LIN {X 0,Y 382.992,Z 182.274,A -85,B 0,C 180,E1 -11850.301,E2 -11850.301} C_VEL
LIN {X 0,Y 383.051,Z 182.269,A -85,B 0,C 180,E1 -11852.698,E2 -11852.698} C_VEL
LIN {X 0,Y 383.046,Z 182.274,A -85,B 0,C 180,E1 -11855.04,E2 -11855.04} C_VEL
LIN {X 0,Y 382.987,Z 182.277,A -85,B 0,C 180,E1 -11858.469,E2 -11858.469} C_VEL
LIN {X 0,Y 383.057,Z 182.266,A -85,B 0,C 180,E1 -11861.827,E2 -11861.827} C_VEL
LIN {X 0,Y 383.104,Z 182.263,A -85,B 0,C 180,E1 -11865.119,E2 -11865.119} C_VEL
LIN {X 0,Y 383.092,Z 182.265,A -85,B 0,C 180,E1 -11868.358,E2 -11868.358} C_VEL
LIN {X 0,Y 383.258,Z 182.242,A -85,B 0,C 180,E1 -11871.976,E2 -11871.976} C_VEL
LIN {X 0,Y 383.192,Z 182.253,A -85,B 0,C 180,E1 -11874.739,E2 -11874.739} C_VEL
LIN {X 0,Y 383.38,Z 182.228,A -85,B 0,C 180,E1 -11877.899,E2 -11877.899} C_VEL
LIN {X 0,Y 383.514,Z 182.212,A -85,B 0,C 180,E1 -11880.001,E2 -11880.001} C_VEL
LIN {X 0,Y 383.24,Z 182.243,A -85,B 0,C 180,E1 -11883.154,E2 -11883.154} C_VEL
LIN {X 0,Y 383.275,Z 182.243,A -85,B 0,C 180,E1 -11886.317,E2 -11886.317} C_VEL
LIN {X 0,Y 383.147,Z 182.256,A -85,B 0,C 180,E1 -11889.503,E2 -11889.503} C_VEL
LIN {X 0,Y 383.121,Z 182.261,A -85,B 0,C 180,E1 -11893.537,E2 -11893.537} C_VEL
LIN {X 0,Y 383.091,Z 182.265,A -85,B 0,C 180,E1 -11897.455,E2 -11897.455} C_VEL
LIN {X 0,Y 383.025,Z 182.27,A -85,B 0,C 180,E1 -11900.648,E2 -11900.648} C_VEL
LIN {X 0,Y 383.03,Z 182.274,A -85,B 0,C 180,E1 -11903.808,E2 -11903.808} C_VEL
LIN {X 0,Y 383.077,Z 182.265,A -85,B 0,C 180,E1 -11906.124,E2 -11906.124} C_VEL
LIN {X 0,Y 382.989,Z 182.278,A -85,B 0,C 180,E1 -11909.701,E2 -11909.701} C_VEL
LIN {X 0,Y 383.001,Z 182.279,A -85,B 0,C 180,E1 -11913.402,E2 -11913.402} C_VEL
LIN {X 0,Y 383.03,Z 182.274,A -85,B 0,C 180,E1 -11916.165,E2 -11916.165} C_VEL
LIN {X 0,Y 382.999,Z 182.279,A -85,B 0,C 180,E1 -11917.905,E2 -11917.905} C_VEL
LIN {X 0,Y 383.44,Z 185.021,A -85,B 0,C 180,E1 -11921.288,E2 -11921.288} C_VEL
LIN {X 0,Y 383.849,Z 188.005,A -85,B 0,C 180,E1 -11924.435,E2 -11924.435} C_VEL
LIN {X 0,Y 384.214,Z 191.062,A -85,B 0,C 180,E1 -11927.407,E2 -11927.407} C_VEL
LIN {X 0,Y 384.098,Z 194.234,A -85,B 0,C 180,E1 -11930.219,E2 -11930.219} C_VEL
LIN {X 0,Y 383.628,Z 198.472,A -85,B 0,C 180,E1 -11933.715,E2 -11933.715} C_VEL
LIN {X 0,Y 383.22,Z 202.206,A -85,B 0,C 180,E1 -11936.621,E2 -11936.621} C_VEL
LIN {X 0,Y 382.801,Z 207.145,A -85,B 0,C 180,E1 -11940.284,E2 -11940.284} C_VEL
LIN {X 0,Y 382.559,Z 210.485,A -85,B 0,C 180,E1 -11942.66,E2 -11942.66} C_VEL
LIN {X 0,Y 382.201,Z 215.542,A -85,B 0,C 180,E1 -11946.138,E2 -11946.138} C_VEL
LIN {X 0,Y 381.971,Z 220.656,A -85,B 0,C 180,E1 -11949.538,E2 -11949.538} C_VEL
LIN {X 0,Y 381.912,Z 223.237,A -85,B 0,C 180,E1 -11951.101,E2 -11951.101} C_VEL
LIN {X 0,Y 383.988,Z 233.513,A -85,B 0,C 180,E1 -11951.545,E2 -11951.545} C_VEL
LIN {X 0,Y 385.643,Z 242.984,A -85,B 0,C 180,E1 -11952.061,E2 -11952.061} C_VEL
LIN {X 0,Y 386.917,Z 251.684,A -85,B 0,C 180,E1 -11952.631,E2 -11952.631} C_VEL
LIN {X 0,Y 387.254,Z 257.307,A -85,B 0,C 180,E1 -11953.025,E2 -11953.025} C_VEL
LIN {X 0,Y 386.212,Z 269.459,A -85,B 0,C 180,E1 -11954.024,E2 -11954.024} C_VEL
LIN {X 0,Y 385.457,Z 278.408,A -85,B 0,C 180,E1 -11954.941,E2 -11954.941} C_VEL
LIN {X 0,Y 384.668,Z 287.294,A -85,B 0,C 180,E1 -11956.04,E2 -11956.04} C_VEL
LIN {X 0,Y 384.084,Z 294.166,A -85,B 0,C 180,E1 -11957.047,E2 -11957.047} C_VEL
LIN {X 0,Y 383.433,Z 300.369,A -85,B 0,C 180,E1 -11958.1,E2 -11958.1} C_VEL
LIN {X 0,Y 382.89,Z 306.911,A -85,B 0,C 180,E1 -11959.423,E2 -11959.423} C_VEL
LIN {X 0,Y 382.464,Z 311.414,A -85,B 0,C 180,E1 -11960.481,E2 -11960.481} C_VEL
LIN {X 0,Y 382.032,Z 316.908,A -85,B 0,C 180,E1 -11962.07,E2 -11962.07} C_VEL
LIN {X 0,Y 381.793,Z 321.235,A -85,B 0,C 180,E1 -11963.659,E2 -11963.659} C_VEL
LIN {X 0,Y 381.684,Z 323.603,A -85,B 0,C 180,E1 -11964.718,E2 -11964.718} C_VEL
LIN {X 0,Y 381.643,Z 325.403,A -85,B 0,C 180,E1 -11965.776,E2 -11965.776} C_VEL
LIN {X 0,Y 381.558,Z 327.847,A -85,B 0,C 180,E1 -11967.889,E2 -11967.889} C_VEL
LIN {X 0,Y 381.591,Z 328.437,A -85,B 0,C 180,E1 -11968.945,E2 -11968.945} C_VEL
LIN {X 0,Y 381.591,Z 328.437,A -85,B 0,C 180,E1 -11971.055,E2 -11971.055} C_VEL
LIN {X 0,Y 381.558,Z 327.847,A -85,B 0,C 180,E1 -11972.111,E2 -11972.111} C_VEL
LIN {X 0,Y 381.643,Z 325.403,A -85,B 0,C 180,E1 -11974.224,E2 -11974.224} C_VEL
LIN {X 0,Y 381.694,Z 322.487,A -85,B 0,C 180,E1 -11975.797,E2 -11975.797} C_VEL
LIN {X 0,Y 381.934,Z 318.462,A -85,B 0,C 180,E1 -11977.401,E2 -11977.401} C_VEL
LIN {X 0,Y 382.305,Z 313.331,A -85,B 0,C 180,E1 -11978.99,E2 -11978.99} C_VEL
LIN {X 0,Y 382.762,Z 308.067,A -85,B 0,C 180,E1 -11980.313,E2 -11980.313} C_VEL
LIN {X 0,Y 383.283,Z 301.745,A -85,B 0,C 180,E1 -11981.636,E2 -11981.636} C_VEL
LIN {X 0,Y 383.901,Z 295.793,A -85,B 0,C 180,E1 -11982.69,E2 -11982.69} C_VEL
LIN {X 0,Y 384.517,Z 288.862,A -85,B 0,C 180,E1 -11983.745,E2 -11983.745} C_VEL
LIN {X 0,Y 385.22,Z 280.677,A -85,B 0,C 180,E1 -11984.798,E2 -11984.798} C_VEL
LIN {X 0,Y 385.952,Z 272.162,A -85,B 0,C 180,E1 -11985.716,E2 -11985.716} C_VEL
LIN {X 0,Y 386.709,Z 263.445,A -85,B 0,C 180,E1 -11986.497,E2 -11986.497} C_VEL
LIN {X 0,Y 387.26,Z 254.506,A -85,B 0,C 180,E1 -11987.164,E2 -11987.164} C_VEL
LIN {X 0,Y 385.889,Z 244.456,A -85,B 0,C 180,E1 -11987.849,E2 -11987.849} C_VEL
LIN {X 0,Y 384.09,Z 233.859,A -85,B 0,C 180,E1 -11988.437,E2 -11988.437} C_VEL
LIN {X 0,Y 381.969,Z 223.863,A -85,B 0,C 180,E1 -11988.879,E2 -11988.879} C_VEL
LIN {X 0,Y 381.882,Z 223.047,A -85,B 0,C 180,E1 -11988.926,E2 -11988.926} C_VEL
LIN {X 0,Y 382.161,Z 217.233,A -85,B 0,C 180,E1 -11992.717,E2 -11992.717} C_VEL
LIN {X 0,Y 382.421,Z 212.16,A -85,B 0,C 180,E1 -11996.171,E2 -11996.171} C_VEL
LIN {X 0,Y 382.686,Z 208.821,A -85,B 0,C 180,E1 -11998.521,E2 -11998.521} C_VEL
LIN {X 0,Y 382.931,Z 205.501,A -85,B 0,C 180,E1 -12000.923,E2 -12000.923} C_VEL
LIN {X 0,Y 383.392,Z 200.573,A -85,B 0,C 180,E1 -12004.629,E2 -12004.629} C_VEL
LIN {X 0,Y 383.871,Z 196.268,A -85,B 0,C 180,E1 -12008.07,E2 -12008.07} C_VEL
LIN {X 0,Y 384.187,Z 192.607,A -85,B 0,C 180,E1 -12011.189,E2 -12011.189} C_VEL
LIN {X 0,Y 384.182,Z 190.641,A -85,B 0,C 180,E1 -12012.967,E2 -12012.967} C_VEL
LIN {X 0,Y 383.789,Z 187.652,A -85,B 0,C 180,E1 -12015.903,E2 -12015.903} C_VEL
LIN {X 0,Y 383.412,Z 184.995,A -85,B 0,C 180,E1 -12018.723,E2 -12018.723} C_VEL
LIN {X 0,Y 383.062,Z 182.677,A -85,B 0,C 180,E1 -12021.406,E2 -12021.406} C_VEL
LIN {X 0,Y 382.992,Z 182.281,A -85,B 0,C 180,E1 -12022.73,E2 -12022.73} C_VEL
LIN {X 0,Y 383.016,Z 182.276,A -85,B 0,C 180,E1 -12025.659,E2 -12025.659} C_VEL
LIN {X 0,Y 382.98,Z 182.278,A -85,B 0,C 180,E1 -12029.081,E2 -12029.081} C_VEL
LIN {X 0,Y 383.054,Z 182.271,A -85,B 0,C 180,E1 -12032.697,E2 -12032.697} C_VEL
LIN {X 0,Y 383.049,Z 182.268,A -85,B 0,C 180,E1 -12035.039,E2 -12035.039} C_VEL
LIN {X 0,Y 382.989,Z 182.28,A -85,B 0,C 180,E1 -12038.468,E2 -12038.468} C_VEL
LIN {X 0,Y 383.059,Z 182.268,A -85,B 0,C 180,E1 -12041.826,E2 -12041.826} C_VEL
LIN {X 0,Y 383.106,Z 182.26,A -85,B 0,C 180,E1 -12045.118,E2 -12045.118} C_VEL
LIN {X 0,Y 383.093,Z 182.265,A -85,B 0,C 180,E1 -12048.357,E2 -12048.357} C_VEL
LIN {X 0,Y 383.258,Z 182.247,A -85,B 0,C 180,E1 -12051.976,E2 -12051.976} C_VEL
LIN {X 0,Y 383.191,Z 182.25,A -85,B 0,C 180,E1 -12054.738,E2 -12054.738} C_VEL
LIN {X 0,Y 383.379,Z 182.231,A -85,B 0,C 180,E1 -12057.898,E2 -12057.898} C_VEL
LIN {X 0,Y 383.514,Z 182.212,A -85,B 0,C 180,E1 -12059.999,E2 -12059.999} C_VEL
LIN {X 0,Y 383.241,Z 182.245,A -85,B 0,C 180,E1 -12063.153,E2 -12063.153} C_VEL
LIN {X 0,Y 383.255,Z 182.242,A -85,B 0,C 180,E1 -12066.635,E2 -12066.635} C_VEL
LIN {X 0,Y 383.146,Z 182.261,A -85,B 0,C 180,E1 -12069.502,E2 -12069.502} C_VEL
LIN {X 0,Y 383.119,Z 182.262,A -85,B 0,C 180,E1 -12073.536,E2 -12073.536} C_VEL
LIN {X 0,Y 383.089,Z 182.266,A -85,B 0,C 180,E1 -12077.454,E2 -12077.454} C_VEL
LIN {X 0,Y 383.022,Z 182.273,A -85,B 0,C 180,E1 -12080.647,E2 -12080.647} C_VEL
LIN {X 0,Y 383.027,Z 182.27,A -85,B 0,C 180,E1 -12083.807,E2 -12083.807} C_VEL
LIN {X 0,Y 383.074,Z 182.264,A -85,B 0,C 180,E1 -12086.123,E2 -12086.123} C_VEL
LIN {X 0,Y 383.043,Z 182.271,A -85,B 0,C 180,E1 -12088.492,E2 -12088.492} C_VEL
LIN {X 0,Y 383.005,Z 182.274,A -85,B 0,C 180,E1 -12092.149,E2 -12092.149} C_VEL
LIN {X 0,Y 383.012,Z 182.278,A -85,B 0,C 180,E1 -12094.668,E2 -12094.668} C_VEL
LIN {X 0,Y 382.997,Z 182.274,A -85,B 0,C 180,E1 -12097.904,E2 -12097.904} C_VEL
LIN {X 0,Y 383.007,Z 182.272,A -85,B 0,C 180,E1 -12101.343,E2 -12101.343} C_VEL
LIN {X 0,Y 382.991,Z 182.28,A -85,B 0,C 180,E1 -12104.303,E2 -12104.303} C_VEL
LIN {X 0,Y 383.004,Z 182.273,A -85,B 0,C 180,E1 -12107.24,E2 -12107.24} C_VEL
LIN {X 0,Y 383.011,Z 182.276,A -85,B 0,C 180,E1 -12110.413,E2 -12110.413} C_VEL
LIN {X 0,Y 383.021,Z 182.277,A -85,B 0,C 180,E1 -12114.045,E2 -12114.045} C_VEL
LIN {X 0,Y 383.032,Z 182.275,A -85,B 0,C 180,E1 -12117.853,E2 -12117.853} C_VEL
LIN {X 0,Y 383.059,Z 182.271,A -85,B 0,C 180,E1 -12121.72,E2 -12121.72} C_VEL
LIN {X 0,Y 383.048,Z 182.268,A -85,B 0,C 180,E1 -12125.04,E2 -12125.04} C_VEL
LIN {X 0,Y 382.992,Z 182.274,A -85,B 0,C 180,E1 -12128.469,E2 -12128.469} C_VEL
LIN {X 0,Y 383.085,Z 182.268,A -85,B 0,C 180,E1 -12131.828,E2 -12131.828} C_VEL
LIN {X 0,Y 383.106,Z 182.265,A -85,B 0,C 180,E1 -12135.118,E2 -12135.118} C_VEL
LIN {X 0,Y 383.094,Z 182.265,A -85,B 0,C 180,E1 -12138.358,E2 -12138.358} C_VEL
LIN {X 0,Y 383.138,Z 182.283,A -85,B 0,C 180,E1 -12139.598,E2 -12139.598} C_VEL
LIN {X 0,Y 383.814,Z 184.561,A -85,B 0,C 180,E1 -12139.95,E2 -12139.95} C_VEL
LIN {X 0,Y 385.348,Z 186.561,A -85,B 0,C 180,E1 -12140.685,E2 -12140.685} C_VEL
LIN {X 0,Y 387.436,Z 187.855,A -85,B 0,C 180,E1 -12141.656,E2 -12141.656} C_VEL
LIN {X 0,Y 388.84,Z 188.564,A -85,B 0,C 180,E1 -12142.402,E2 -12142.402} C_VEL
LIN {X 0,Y 389.96,Z 190.834,A -85,B 0,C 180,E1 -12143.142,E2 -12143.142} C_VEL
LIN {X 0,Y 391.789,Z 192.993,A -85,B 0,C 180,E1 -12144.467,E2 -12144.467} C_VEL
LIN {X 0,Y 393.422,Z 194.061,A -85,B 0,C 180,E1 -12145.902,E2 -12145.902} C_VEL
LIN {X 0,Y 394.945,Z 194.431,A -85,B 0,C 180,E1 -12147.96,E2 -12147.96} C_VEL
LIN {X 0,Y 395.509,Z 194.494,A -85,B 0,C 180,E1 -12150,E2 -12150} C_VEL
LIN {X 0,Y 394.945,Z 194.431,A -85,B 0,C 180,E1 -12152.04,E2 -12152.04} C_VEL
LIN {X 0,Y 393.422,Z 194.061,A -85,B 0,C 180,E1 -12154.098,E2 -12154.098} C_VEL
LIN {X 0,Y 391.446,Z 192.7,A -85,B 0,C 180,E1 -12155.796,E2 -12155.796} C_VEL
LIN {X 0,Y 389.552,Z 190.154,A -85,B 0,C 180,E1 -12157.135,E2 -12157.135} C_VEL
LIN {X 0,Y 388.788,Z 188.398,A -85,B 0,C 180,E1 -12157.634,E2 -12157.634} C_VEL
LIN {X 0,Y 385.958,Z 187.055,A -85,B 0,C 180,E1 -12159.036,E2 -12159.036} C_VEL
LIN {X 0,Y 384.054,Z 184.967,A -85,B 0,C 180,E1 -12159.938,E2 -12159.938} C_VEL
LIN {X 0,Y 383.253,Z 182.924,A -85,B 0,C 180,E1 -12160.332,E2 -12160.332} C_VEL
LIN {X 0,Y 383.121,Z 182.263,A -85,B 0,C 180,E1 -12160.436,E2 -12160.436} C_VEL
LIN {X 0,Y 383.123,Z 182.262,A -85,B 0,C 180,E1 -12163.796,E2 -12163.796} C_VEL
LIN {X 0,Y 383.091,Z 182.267,A -85,B 0,C 180,E1 -12167.455,E2 -12167.455} C_VEL
LIN {X 0,Y 383.03,Z 182.273,A -85,B 0,C 180,E1 -12170.649,E2 -12170.649} C_VEL
LIN {X 0,Y 383.029,Z 182.271,A -85,B 0,C 180,E1 -12173.807,E2 -12173.807} C_VEL
LIN {X 0,Y 383.052,Z 182.267,A -85,B 0,C 180,E1 -12177.302,E2 -12177.302} C_VEL
LIN {X 0,Y 382.991,Z 182.275,A -85,B 0,C 180,E1 -12180.917,E2 -12180.917} C_VEL
LIN {X 0,Y 383.013,Z 182.274,A -85,B 0,C 180,E1 -12184.34,E2 -12184.34} C_VEL
LIN {X 0,Y 382.994,Z 182.275,A -85,B 0,C 180,E1 -12185.374,E2 -12185.374} C_VEL
LIN {X 0,Y 382.353,Z 182.361,A -85,B 0,C 180,E1 -12186.252,E2 -12186.252} C_VEL
LIN {X 0,Y 379.545,Z 182.717,A -85,B 0,C 180,E1 -12187.68,E2 -12187.68} C_VEL
LIN {X 0,Y 377.141,Z 183.016,A -85,B 0,C 180,E1 -12188.835,E2 -12188.835} C_VEL
LIN {X 0,Y 376.086,Z 183.142,A -85,B 0,C 180,E1 -12189.727,E2 -12189.727} C_VEL
LIN {X 0,Y 375.988,Z 183.151,A -85,B 0,C 180,E1 -12190.029,E2 -12190.029} C_VEL
LIN {X 0,Y 375.934,Z 183.159,A -85,B 0,C 180,E1 -12193.765,E2 -12193.765} C_VEL
LIN {X 0,Y 375.955,Z 183.156,A -85,B 0,C 180,E1 -12197.704,E2 -12197.704} C_VEL
LIN {X 0,Y 375.963,Z 183.15,A -85,B 0,C 180,E1 -12200.538,E2 -12200.538} C_VEL
LIN {X 0,Y 375.959,Z 183.156,A -85,B 0,C 180,E1 -12203.495,E2 -12203.495} C_VEL
LIN {X 0,Y 375.954,Z 183.152,A -85,B 0,C 180,E1 -12205.889,E2 -12205.889} C_VEL
LIN {X 0,Y 375.962,Z 183.152,A -85,B 0,C 180,E1 -12209.688,E2 -12209.688} C_VEL
LIN {X 0,Y 375.996,Z 183.146,A -85,B 0,C 180,E1 -12212.142,E2 -12212.142} C_VEL
LIN {X 0,Y 376,Z 183.147,A -85,B 0,C 180,E1 -12214.539,E2 -12214.539} C_VEL
LIN {X 0,Y 375.957,Z 183.151,A -85,B 0,C 180,E1 -12218.046,E2 -12218.046} C_VEL
LIN {X 0,Y 376.003,Z 183.146,A -85,B 0,C 180,E1 -12221.474,E2 -12221.474} C_VEL
LIN {X 0,Y 376.052,Z 183.145,A -85,B 0,C 180,E1 -12224.833,E2 -12224.833} C_VEL
LIN {X 0,Y 376.044,Z 183.141,A -85,B 0,C 180,E1 -12228.137,E2 -12228.137} C_VEL
LIN {X 0,Y 376.214,Z 183.119,A -85,B 0,C 180,E1 -12231.919,E2 -12231.919} C_VEL
LIN {X 0,Y 376.165,Z 183.129,A -85,B 0,C 180,E1 -12234.64,E2 -12234.64} C_VEL
LIN {X 0,Y 376.346,Z 183.104,A -85,B 0,C 180,E1 -12237.86,E2 -12237.86} C_VEL
LIN {X 0,Y 376.483,Z 183.088,A -85,B 0,C 180,E1 -12240.001,E2 -12240.001} C_VEL
LIN {X 0,Y 376.179,Z 183.123,A -85,B 0,C 180,E1 -12243.214,E2 -12243.214} C_VEL
LIN {X 0,Y 376.233,Z 183.119,A -85,B 0,C 180,E1 -12246.436,E2 -12246.436} C_VEL
LIN {X 0,Y 376.114,Z 183.134,A -85,B 0,C 180,E1 -12249.682,E2 -12249.682} C_VEL
LIN {X 0,Y 376.085,Z 183.138,A -85,B 0,C 180,E1 -12253.658,E2 -12253.658} C_VEL
LIN {X 0,Y 376.039,Z 183.145,A -85,B 0,C 180,E1 -12257.608,E2 -12257.608} C_VEL
LIN {X 0,Y 375.975,Z 183.149,A -85,B 0,C 180,E1 -12260.833,E2 -12260.833} C_VEL
LIN {X 0,Y 375.991,Z 183.147,A -85,B 0,C 180,E1 -12264.282,E2 -12264.282} C_VEL
LIN {X 0,Y 376.017,Z 183.143,A -85,B 0,C 180,E1 -12266.653,E2 -12266.653} C_VEL
LIN {X 0,Y 375.962,Z 183.15,A -85,B 0,C 180,E1 -12270.313,E2 -12270.313} C_VEL
LIN {X 0,Y 375.958,Z 183.155,A -85,B 0,C 180,E1 -12274.112,E2 -12274.112} C_VEL
LIN {X 0,Y 375.951,Z 183.158,A -85,B 0,C 180,E1 -12276.742,E2 -12276.742} C_VEL
LIN {X 0,Y 376.023,Z 183.591,A -85,B 0,C 180,E1 -12278.281,E2 -12278.281} C_VEL
LIN {X 0,Y 376.47,Z 186.515,A -85,B 0,C 180,E1 -12281.693,E2 -12281.693} C_VEL
LIN {X 0,Y 376.906,Z 189.765,A -85,B 0,C 180,E1 -12285.119,E2 -12285.119} C_VEL
LIN {X 0,Y 377.168,Z 192.589,A -85,B 0,C 180,E1 -12287.871,E2 -12287.871} C_VEL
LIN {X 0,Y 376.988,Z 195.718,A -85,B 0,C 180,E1 -12290.666,E2 -12290.666} C_VEL
LIN {X 0,Y 376.631,Z 198.928,A -85,B 0,C 180,E1 -12293.359,E2 -12293.359} C_VEL
LIN {X 0,Y 376.25,Z 202.125,A -85,B 0,C 180,E1 -12295.919,E2 -12295.919} C_VEL
LIN {X 0,Y 375.826,Z 207.042,A -85,B 0,C 180,E1 -12299.676,E2 -12299.676} C_VEL
LIN {X 0,Y 375.556,Z 210.367,A -85,B 0,C 180,E1 -12302.106,E2 -12302.106} C_VEL
LIN {X 0,Y 375.158,Z 215.391,A -85,B 0,C 180,E1 -12305.661,E2 -12305.661} C_VEL
LIN {X 0,Y 375.007,Z 218.771,A -85,B 0,C 180,E1 -12307.987,E2 -12307.987} C_VEL
LIN {X 0,Y 374.836,Z 222.855,A -85,B 0,C 180,E1 -12310.722,E2 -12310.722} C_VEL
LIN {X 0,Y 377.036,Z 233.737,A -85,B 0,C 180,E1 -12311.209,E2 -12311.209} C_VEL
LIN {X 0,Y 378.619,Z 242.764,A -85,B 0,C 180,E1 -12311.717,E2 -12311.717} C_VEL
LIN {X 0,Y 379.924,Z 251.828,A -85,B 0,C 180,E1 -12312.326,E2 -12312.326} C_VEL
LIN {X 0,Y 380.448,Z 257.164,A -85,B 0,C 180,E1 -12312.717,E2 -12312.717} C_VEL
LIN {X 0,Y 379.377,Z 269.247,A -85,B 0,C 180,E1 -12313.729,E2 -12313.729} C_VEL
LIN {X 0,Y 378.587,Z 278.196,A -85,B 0,C 180,E1 -12314.661,E2 -12314.661} C_VEL
LIN {X 0,Y 377.873,Z 285.861,A -85,B 0,C 180,E1 -12315.609,E2 -12315.609} C_VEL
LIN {X 0,Y 377.152,Z 293.954,A -85,B 0,C 180,E1 -12316.805,E2 -12316.805} C_VEL
LIN {X 0,Y 376.469,Z 300.157,A -85,B 0,C 180,E1 -12317.877,E2 -12317.877} C_VEL
LIN {X 0,Y 375.853,Z 306.698,A -85,B 0,C 180,E1 -12319.223,E2 -12319.223} C_VEL
LIN {X 0,Y 375.451,Z 311.202,A -85,B 0,C 180,E1 -12320.301,E2 -12320.301} C_VEL
LIN {X 0,Y 374.964,Z 316.695,A -85,B 0,C 180,E1 -12321.919,E2 -12321.919} C_VEL
LIN {X 0,Y 374.72,Z 321.023,A -85,B 0,C 180,E1 -12323.539,E2 -12323.539} C_VEL
LIN {X 0,Y 374.591,Z 323.391,A -85,B 0,C 180,E1 -12324.617,E2 -12324.617} C_VEL
LIN {X 0,Y 374.57,Z 325.192,A -85,B 0,C 180,E1 -12325.696,E2 -12325.696} C_VEL
LIN {X 0,Y 374.458,Z 327.636,A -85,B 0,C 180,E1 -12327.849,E2 -12327.849} C_VEL
LIN {X 0,Y 374.492,Z 328.226,A -85,B 0,C 180,E1 -12328.925,E2 -12328.925} C_VEL
LIN {X 0,Y 374.492,Z 328.226,A -85,B 0,C 180,E1 -12331.075,E2 -12331.075} C_VEL
LIN {X 0,Y 374.458,Z 327.636,A -85,B 0,C 180,E1 -12332.151,E2 -12332.151} C_VEL
LIN {X 0,Y 374.571,Z 325.192,A -85,B 0,C 180,E1 -12334.304,E2 -12334.304} C_VEL
LIN {X 0,Y 374.592,Z 323.391,A -85,B 0,C 180,E1 -12335.383,E2 -12335.383} C_VEL
LIN {X 0,Y 374.77,Z 319.781,A -85,B 0,C 180,E1 -12337.001,E2 -12337.001} C_VEL
LIN {X 0,Y 375.102,Z 315.034,A -85,B 0,C 180,E1 -12338.62,E2 -12338.62} C_VEL
LIN {X 0,Y 375.631,Z 309.01,A -85,B 0,C 180,E1 -12340.238,E2 -12340.238} C_VEL
LIN {X 0,Y 376.18,Z 302.91,A -85,B 0,C 180,E1 -12341.586,E2 -12341.586} C_VEL
LIN {X 0,Y 376.78,Z 297.208,A -85,B 0,C 180,E1 -12342.66,E2 -12342.66} C_VEL
LIN {X 0,Y 377.594,Z 288.65,A -85,B 0,C 180,E1 -12344.002,E2 -12344.002} C_VEL
LIN {X 0,Y 378.322,Z 280.465,A -85,B 0,C 180,E1 -12345.074,E2 -12345.074} C_VEL
LIN {X 0,Y 379.122,Z 271.951,A -85,B 0,C 180,E1 -12346.006,E2 -12346.006} C_VEL
LIN {X 0,Y 379.889,Z 263.233,A -85,B 0,C 180,E1 -12346.802,E2 -12346.802} C_VEL
LIN {X 0,Y 380.447,Z 255.846,A -85,B 0,C 180,E1 -12347.374,E2 -12347.374} C_VEL
LIN {X 0,Y 378.927,Z 244.579,A -85,B 0,C 180,E1 -12348.17,E2 -12348.17} C_VEL
LIN {X 0,Y 377.133,Z 234.279,A -85,B 0,C 180,E1 -12348.764,E2 -12348.764} C_VEL
LIN {X 0,Y 374.92,Z 223.683,A -85,B 0,C 180,E1 -12349.247,E2 -12349.247} C_VEL
LIN {X 0,Y 374.843,Z 222.829,A -85,B 0,C 180,E1 -12349.296,E2 -12349.296} C_VEL
LIN {X 0,Y 375.117,Z 216.798,A -85,B 0,C 180,E1 -12353.358,E2 -12353.358} C_VEL
LIN {X 0,Y 375.389,Z 212.026,A -85,B 0,C 180,E1 -12356.7,E2 -12356.7} C_VEL
LIN {X 0,Y 375.823,Z 207.042,A -85,B 0,C 180,E1 -12360.325,E2 -12360.325} C_VEL
LIN {X 0,Y 376.249,Z 202.125,A -85,B 0,C 180,E1 -12364.081,E2 -12364.081} C_VEL
LIN {X 0,Y 376.634,Z 198.901,A -85,B 0,C 180,E1 -12366.663,E2 -12366.663} C_VEL
LIN {X 0,Y 377.086,Z 194.756,A -85,B 0,C 180,E1 -12370.168,E2 -12370.168} C_VEL
LIN {X 0,Y 377.164,Z 192.57,A -85,B 0,C 180,E1 -12372.129,E2 -12372.129} C_VEL
LIN {X 0,Y 376.867,Z 189.497,A -85,B 0,C 180,E1 -12375.124,E2 -12375.124} C_VEL
LIN {X 0,Y 376.447,Z 186.513,A -85,B 0,C 180,E1 -12378.31,E2 -12378.31} C_VEL
LIN {X 0,Y 376.023,Z 183.598,A -85,B 0,C 180,E1 -12381.719,E2 -12381.719} C_VEL
LIN {X 0,Y 375.961,Z 183.151,A -85,B 0,C 180,E1 -12383.495,E2 -12383.495} C_VEL
LIN {X 0,Y 375.958,Z 183.154,A -85,B 0,C 180,E1 -12385.888,E2 -12385.888} C_VEL
LIN {X 0,Y 375.962,Z 183.15,A -85,B 0,C 180,E1 -12389.687,E2 -12389.687} C_VEL
LIN {X 0,Y 376.017,Z 183.143,A -85,B 0,C 180,E1 -12393.347,E2 -12393.347} C_VEL
LIN {X 0,Y 375.993,Z 183.148,A -85,B 0,C 180,E1 -12396.888,E2 -12396.888} C_VEL
LIN {X 0,Y 375.995,Z 183.152,A -85,B 0,C 180,E1 -12400.339,E2 -12400.339} C_VEL
LIN {X 0,Y 376.025,Z 183.144,A -85,B 0,C 180,E1 -12403.718,E2 -12403.718} C_VEL
LIN {X 0,Y 376.099,Z 183.133,A -85,B 0,C 180,E1 -12407.041,E2 -12407.041} C_VEL
LIN {X 0,Y 376.114,Z 183.134,A -85,B 0,C 180,E1 -12410.318,E2 -12410.318} C_VEL
LIN {X 0,Y 376.233,Z 183.119,A -85,B 0,C 180,E1 -12413.564,E2 -12413.564} C_VEL
LIN {X 0,Y 376.345,Z 183.108,A -85,B 0,C 180,E1 -12417.859,E2 -12417.859} C_VEL
LIN {X 0,Y 376.483,Z 183.088,A -85,B 0,C 180,E1 -12419.999,E2 -12419.999} C_VEL
LIN {X 0,Y 376.18,Z 183.125,A -85,B 0,C 180,E1 -12423.212,E2 -12423.212} C_VEL
LIN {X 0,Y 376.22,Z 183.118,A -85,B 0,C 180,E1 -12426.624,E2 -12426.624} C_VEL
LIN {X 0,Y 376.113,Z 183.135,A -85,B 0,C 180,E1 -12429.681,E2 -12429.681} C_VEL
LIN {X 0,Y 376.084,Z 183.137,A -85,B 0,C 180,E1 -12433.657,E2 -12433.657} C_VEL
LIN {X 0,Y 376.037,Z 183.143,A -85,B 0,C 180,E1 -12437.606,E2 -12437.606} C_VEL
LIN {X 0,Y 375.972,Z 183.153,A -85,B 0,C 180,E1 -12440.832,E2 -12440.832} C_VEL
LIN {X 0,Y 375.988,Z 183.147,A -85,B 0,C 180,E1 -12444.281,E2 -12444.281} C_VEL
LIN {X 0,Y 376.014,Z 183.147,A -85,B 0,C 180,E1 -12446.652,E2 -12446.652} C_VEL
LIN {X 0,Y 375.97,Z 183.153,A -85,B 0,C 180,E1 -12449.078,E2 -12449.078} C_VEL
LIN {X 0,Y 375.943,Z 183.158,A -85,B 0,C 180,E1 -12452.828,E2 -12452.828} C_VEL
LIN {X 0,Y 375.952,Z 183.152,A -85,B 0,C 180,E1 -12455.415,E2 -12455.415} C_VEL
LIN {X 0,Y 375.972,Z 183.152,A -85,B 0,C 180,E1 -12458.271,E2 -12458.271} C_VEL
LIN {X 0,Y 375.954,Z 183.151,A -85,B 0,C 180,E1 -12461.605,E2 -12461.605} C_VEL
LIN {X 0,Y 375.921,Z 183.155,A -85,B 0,C 180,E1 -12465.269,E2 -12465.269} C_VEL
LIN {X 0,Y 375.929,Z 183.159,A -85,B 0,C 180,E1 -12468.399,E2 -12468.399} C_VEL
LIN {X 0,Y 375.971,Z 183.151,A -85,B 0,C 180,E1 -12471.729,E2 -12471.729} C_VEL
LIN {X 0,Y 375.975,Z 183.149,A -85,B 0,C 180,E1 -12475.333,E2 -12475.333} C_VEL
LIN {X 0,Y 375.971,Z 183.151,A -85,B 0,C 180,E1 -12478.44,E2 -12478.44} C_VEL
LIN {X 0,Y 375.998,Z 183.149,A -85,B 0,C 180,E1 -12482.142,E2 -12482.142} C_VEL
LIN {X 0,Y 376.002,Z 183.145,A -85,B 0,C 180,E1 -12484.539,E2 -12484.539} C_VEL
LIN {X 0,Y 375.961,Z 183.153,A -85,B 0,C 180,E1 -12488.046,E2 -12488.046} C_VEL
LIN {X 0,Y 376.02,Z 183.148,A -85,B 0,C 180,E1 -12491.474,E2 -12491.474} C_VEL
LIN {X 0,Y 376.055,Z 183.144,A -85,B 0,C 180,E1 -12494.833,E2 -12494.833} C_VEL
LIN {X 0,Y 376.117,Z 183.315,A -85,B 0,C 180,E1 -12497.317,E2 -12497.317} C_VEL
LIN {X 0,Y 376.774,Z 185.472,A -85,B 0,C 180,E1 -12497.613,E2 -12497.613} C_VEL
LIN {X 0,Y 378.391,Z 187.585,A -85,B 0,C 180,E1 -12498.211,E2 -12498.211} C_VEL
LIN {X 0,Y 380.855,Z 188.996,A -85,B 0,C 180,E1 -12499.097,E2 -12499.097} C_VEL
LIN {X 0,Y 381.348,Z 189.793,A -85,B 0,C 180,E1 -12499.313,E2 -12499.313} C_VEL
LIN {X 0,Y 382.988,Z 192.386,A -85,B 0,C 180,E1 -12500.027,E2 -12500.027} C_VEL
LIN {X 0,Y 385.299,Z 194.35,A -85,B 0,C 180,E1 -12501.081,E2 -12501.081} C_VEL
LIN {X 0,Y 387.405,Z 195.44,A -85,B 0,C 180,E1 -12502.125,E2 -12502.125} C_VEL
LIN {X 0,Y 388.935,Z 197.999,A -85,B 0,C 180,E1 -12503.079,E2 -12503.079} C_VEL
LIN {X 0,Y 390.889,Z 200.077,A -85,B 0,C 180,E1 -12504.454,E2 -12504.454} C_VEL
LIN {X 0,Y 392.534,Z 201.093,A -85,B 0,C 180,E1 -12505.893,E2 -12505.893} C_VEL
LIN {X 0,Y 394.082,Z 201.477,A -85,B 0,C 180,E1 -12507.956,E2 -12507.956} C_VEL
LIN {X 0,Y 394.645,Z 201.533,A -85,B 0,C 180,E1 -12510,E2 -12510} C_VEL
LIN {X 0,Y 394.082,Z 201.477,A -85,B 0,C 180,E1 -12512.044,E2 -12512.044} C_VEL
LIN {X 0,Y 392.534,Z 201.093,A -85,B 0,C 180,E1 -12514.107,E2 -12514.107} C_VEL
LIN {X 0,Y 390.529,Z 199.798,A -85,B 0,C 180,E1 -12515.81,E2 -12515.81} C_VEL
LIN {X 0,Y 388.397,Z 197.203,A -85,B 0,C 180,E1 -12517.277,E2 -12517.277} C_VEL
LIN {X 0,Y 387.178,Z 195.131,A -85,B 0,C 180,E1 -12518.008,E2 -12518.008} C_VEL
LIN {X 0,Y 384.673,Z 193.95,A -85,B 0,C 180,E1 -12519.199,E2 -12519.199} C_VEL
LIN {X 0,Y 382.482,Z 191.776,A -85,B 0,C 180,E1 -12520.187,E2 -12520.187} C_VEL
LIN {X 0,Y 381.134,Z 189.202,A -85,B 0,C 180,E1 -12520.792,E2 -12520.792} C_VEL
LIN {X 0,Y 378.391,Z 187.585,A -85,B 0,C 180,E1 -12521.789,E2 -12521.789} C_VEL
LIN {X 0,Y 376.728,Z 185.375,A -85,B 0,C 180,E1 -12522.405,E2 -12522.405} C_VEL
LIN {X 0,Y 376.108,Z 183.138,A -85,B 0,C 180,E1 -12522.717,E2 -12522.717} C_VEL
LIN {X 0,Y 376.025,Z 183.147,A -85,B 0,C 180,E1 -12526.281,E2 -12526.281} C_VEL
LIN {X 0,Y 375.996,Z 183.148,A -85,B 0,C 180,E1 -12529.66,E2 -12529.66} C_VEL
LIN {X 0,Y 375.991,Z 183.147,A -85,B 0,C 180,E1 -12533.667,E2 -12533.667} C_VEL
LIN {X 0,Y 376.015,Z 183.145,A -85,B 0,C 180,E1 -12536.652,E2 -12536.652} C_VEL
LIN {X 0,Y 375.972,Z 183.149,A -85,B 0,C 180,E1 -12539.078,E2 -12539.078} C_VEL
LIN {X 0,Y 375.953,Z 183.151,A -85,B 0,C 180,E1 -12542.828,E2 -12542.828} C_VEL
LIN {X 0,Y 375.953,Z 183.153,A -85,B 0,C 180,E1 -12545.415,E2 -12545.415} C_VEL
LIN {X 0,Y 375.972,Z 183.151,A -85,B 0,C 180,E1 -12548.271,E2 -12548.271} C_VEL
LIN {X 0,Y 375.988,Z 183.151,A -85,B 0,C 180,E1 -12550.029,E2 -12550.029} C_VEL
LIN {X 0,Y 375.276,Z 183.236,A -85,B 0,C 180,E1 -12550.922,E2 -12550.922} C_VEL
LIN {X 0,Y 372.37,Z 183.598,A -85,B 0,C 180,E1 -12552.375,E2 -12552.375} C_VEL
LIN {X 0,Y 369.949,Z 183.904,A -85,B 0,C 180,E1 -12553.549,E2 -12553.549} C_VEL
LIN {X 0,Y 368.939,Z 184.025,A -85,B 0,C 180,E1 -12554.458,E2 -12554.458} C_VEL
LIN {X 0,Y 368.871,Z 184.033,A -85,B 0,C 180,E1 -12554.765,E2 -12554.765} C_VEL
LIN {X 0,Y 368.904,Z 184.03,A -85,B 0,C 180,E1 -12558.181,E2 -12558.181} C_VEL
LIN {X 0,Y 368.908,Z 184.034,A -85,B 0,C 180,E1 -12561.359,E2 -12561.359} C_VEL
LIN {X 0,Y 368.931,Z 184.03,A -85,B 0,C 180,E1 -12565.147,E2 -12565.147} C_VEL
LIN {X 0,Y 368.923,Z 184.031,A -85,B 0,C 180,E1 -12569.047,E2 -12569.047} C_VEL
LIN {X 0,Y 368.981,Z 184.022,A -85,B 0,C 180,E1 -12571.565,E2 -12571.565} C_VEL
LIN {X 0,Y 368.951,Z 184.028,A -85,B 0,C 180,E1 -12575.225,E2 -12575.225} C_VEL
LIN {X 0,Y 368.932,Z 184.032,A -85,B 0,C 180,E1 -12578.974,E2 -12578.974} C_VEL
LIN {X 0,Y 368.985,Z 184.02,A -85,B 0,C 180,E1 -12582.258,E2 -12582.258} C_VEL
LIN {X 0,Y 369.031,Z 184.015,A -85,B 0,C 180,E1 -12586.228,E2 -12586.228} C_VEL
LIN {X 0,Y 369.062,Z 184.011,A -85,B 0,C 180,E1 -12590.132,E2 -12590.132} C_VEL
LIN {X 0,Y 369.195,Z 183.993,A -85,B 0,C 180,E1 -12593.442,E2 -12593.442} C_VEL
LIN {X 0,Y 369.311,Z 183.98,A -85,B 0,C 180,E1 -12597.819,E2 -12597.819} C_VEL
LIN {X 0,Y 369.453,Z 183.964,A -85,B 0,C 180,E1 -12600.001,E2 -12600.001} C_VEL
LIN {X 0,Y 369.311,Z 183.984,A -85,B 0,C 180,E1 -12602.182,E2 -12602.182} C_VEL
LIN {X 0,Y 369.194,Z 183.995,A -85,B 0,C 180,E1 -12606.559,E2 -12606.559} C_VEL
LIN {X 0,Y 369.063,Z 184.014,A -85,B 0,C 180,E1 -12609.869,E2 -12609.869} C_VEL
LIN {X 0,Y 369.033,Z 184.018,A -85,B 0,C 180,E1 -12613.773,E2 -12613.773} C_VEL
LIN {X 0,Y 368.998,Z 184.024,A -85,B 0,C 180,E1 -12617.769,E2 -12617.769} C_VEL
LIN {X 0,Y 368.926,Z 184.028,A -85,B 0,C 180,E1 -12621.22,E2 -12621.22} C_VEL
LIN {X 0,Y 368.955,Z 184.023,A -85,B 0,C 180,E1 -12624.776,E2 -12624.776} C_VEL
LIN {X 0,Y 368.96,Z 184.025,A -85,B 0,C 180,E1 -12627.204,E2 -12627.204} C_VEL
LIN {X 0,Y 368.927,Z 184.028,A -85,B 0,C 180,E1 -12630.954,E2 -12630.954} C_VEL
LIN {X 0,Y 368.927,Z 184.032,A -85,B 0,C 180,E1 -12635.002,E2 -12635.002} C_VEL
LIN {X 0,Y 368.932,Z 184.199,A -85,B 0,C 180,E1 -12637.56,E2 -12637.56} C_VEL
LIN {X 0,Y 369.295,Z 186.54,A -85,B 0,C 180,E1 -12640.428,E2 -12640.428} C_VEL
LIN {X 0,Y 369.713,Z 189.523,A -85,B 0,C 180,E1 -12643.752,E2 -12643.752} C_VEL
LIN {X 0,Y 370.091,Z 192.578,A -85,B 0,C 180,E1 -12646.872,E2 -12646.872} C_VEL
LIN {X 0,Y 370.058,Z 195.691,A -85,B 0,C 180,E1 -12649.781,E2 -12649.781} C_VEL
LIN {X 0,Y 369.614,Z 199.396,A -85,B 0,C 180,E1 -12652.998,E2 -12652.998} C_VEL
LIN {X 0,Y 369.105,Z 203.672,A -85,B 0,C 180,E1 -12656.484,E2 -12656.484} C_VEL
LIN {X 0,Y 368.666,Z 208.579,A -85,B 0,C 180,E1 -12660.288,E2 -12660.288} C_VEL
LIN {X 0,Y 368.3,Z 213.278,A -85,B 0,C 180,E1 -12663.75,E2 -12663.75} C_VEL
LIN {X 0,Y 367.948,Z 218.597,A -85,B 0,C 180,E1 -12667.542,E2 -12667.542} C_VEL
LIN {X 0,Y 367.76,Z 222.609,A -85,B 0,C 180,E1 -12670.318,E2 -12670.318} C_VEL
LIN {X 0,Y 370.839,Z 237.835,A -85,B 0,C 180,E1 -12671.063,E2 -12671.063} C_VEL
LIN {X 0,Y 372.833,Z 250.677,A -85,B 0,C 180,E1 -12671.913,E2 -12671.913} C_VEL
LIN {X 0,Y 373.587,Z 258.125,A -85,B 0,C 180,E1 -12672.483,E2 -12672.483} C_VEL
LIN {X 0,Y 372.554,Z 269.036,A -85,B 0,C 180,E1 -12673.422,E2 -12673.422} C_VEL
LIN {X 0,Y 371.714,Z 277.984,A -85,B 0,C 180,E1 -12674.37,E2 -12674.37} C_VEL
LIN {X 0,Y 370.942,Z 286.001,A -85,B 0,C 180,E1 -12675.386,E2 -12675.386} C_VEL
LIN {X 0,Y 370.226,Z 293.743,A -85,B 0,C 180,E1 -12676.553,E2 -12676.553} C_VEL
LIN {X 0,Y 369.518,Z 299.945,A -85,B 0,C 180,E1 -12677.645,E2 -12677.645} C_VEL
LIN {X 0,Y 368.831,Z 306.485,A -85,B 0,C 180,E1 -12679.015,E2 -12679.015} C_VEL
LIN {X 0,Y 368.414,Z 310.99,A -85,B 0,C 180,E1 -12680.114,E2 -12680.114} C_VEL
LIN {X 0,Y 367.911,Z 316.483,A -85,B 0,C 180,E1 -12681.763,E2 -12681.763} C_VEL
LIN {X 0,Y 367.644,Z 320.811,A -85,B 0,C 180,E1 -12683.414,E2 -12683.414} C_VEL
LIN {X 0,Y 367.507,Z 323.179,A -85,B 0,C 180,E1 -12684.513,E2 -12684.513} C_VEL
LIN {X 0,Y 367.476,Z 324.98,A -85,B 0,C 180,E1 -12685.613,E2 -12685.613} C_VEL
LIN {X 0,Y 367.359,Z 327.424,A -85,B 0,C 180,E1 -12687.807,E2 -12687.807} C_VEL
LIN {X 0,Y 367.392,Z 328.015,A -85,B 0,C 180,E1 -12688.904,E2 -12688.904} C_VEL
LIN {X 0,Y 367.392,Z 328.015,A -85,B 0,C 180,E1 -12691.096,E2 -12691.096} C_VEL
LIN {X 0,Y 367.359,Z 327.424,A -85,B 0,C 180,E1 -12692.193,E2 -12692.193} C_VEL
LIN {X 0,Y 367.477,Z 324.98,A -85,B 0,C 180,E1 -12694.387,E2 -12694.387} C_VEL
LIN {X 0,Y 367.552,Z 321.85,A -85,B 0,C 180,E1 -12696.117,E2 -12696.117} C_VEL
LIN {X 0,Y 367.793,Z 318.038,A -85,B 0,C 180,E1 -12697.687,E2 -12697.687} C_VEL
LIN {X 0,Y 368.231,Z 312.906,A -85,B 0,C 180,E1 -12699.336,E2 -12699.336} C_VEL
LIN {X 0,Y 368.75,Z 307.643,A -85,B 0,C 180,E1 -12700.709,E2 -12700.709} C_VEL
LIN {X 0,Y 369.337,Z 301.321,A -85,B 0,C 180,E1 -12702.082,E2 -12702.082} C_VEL
LIN {X 0,Y 370.031,Z 295.37,A -85,B 0,C 180,E1 -12703.174,E2 -12703.174} C_VEL
LIN {X 0,Y 370.844,Z 287.174,A -85,B 0,C 180,E1 -12704.447,E2 -12704.447} C_VEL
LIN {X 0,Y 371.565,Z 279.118,A -85,B 0,C 180,E1 -12705.496,E2 -12705.496} C_VEL
LIN {X 0,Y 372.415,Z 270.387,A -85,B 0,C 180,E1 -12706.443,E2 -12706.443} C_VEL
LIN {X 0,Y 373.245,Z 261.389,A -85,B 0,C 180,E1 -12707.251,E2 -12707.251} C_VEL
LIN {X 0,Y 373.467,Z 255.762,A -85,B 0,C 180,E1 -12707.7,E2 -12707.7} C_VEL
LIN {X 0,Y 371.986,Z 244.811,A -85,B 0,C 180,E1 -12708.497,E2 -12708.497} C_VEL
LIN {X 0,Y 370.095,Z 233.941,A -85,B 0,C 180,E1 -12709.139,E2 -12709.139} C_VEL
LIN {X 0,Y 367.824,Z 223.374,A -85,B 0,C 180,E1 -12709.636,E2 -12709.636} C_VEL
LIN {X 0,Y 367.763,Z 222.614,A -85,B 0,C 180,E1 -12709.679,E2 -12709.679} C_VEL
LIN {X 0,Y 368.053,Z 216.909,A -85,B 0,C 180,E1 -12713.64,E2 -12713.64} C_VEL
LIN {X 0,Y 368.383,Z 211.893,A -85,B 0,C 180,E1 -12717.249,E2 -12717.249} C_VEL
LIN {X 0,Y 368.82,Z 206.931,A -85,B 0,C 180,E1 -12720.963,E2 -12720.963} C_VEL
LIN {X 0,Y 369.328,Z 202.05,A -85,B 0,C 180,E1 -12724.811,E2 -12724.811} C_VEL
LIN {X 0,Y 369.675,Z 198.838,A -85,B 0,C 180,E1 -12727.47,E2 -12727.47} C_VEL
LIN {X 0,Y 370.083,Z 195.28,A -85,B 0,C 180,E1 -12730.569,E2 -12730.569} C_VEL
LIN {X 0,Y 370.09,Z 192.555,A -85,B 0,C 180,E1 -12733.128,E2 -12733.128} C_VEL
LIN {X 0,Y 369.699,Z 189.51,A -85,B 0,C 180,E1 -12736.251,E2 -12736.251} C_VEL
LIN {X 0,Y 369.283,Z 186.45,A -85,B 0,C 180,E1 -12739.678,E2 -12739.678} C_VEL
LIN {X 0,Y 368.917,Z 184.2,A -85,B 0,C 180,E1 -12742.438,E2 -12742.438} C_VEL
LIN {X 0,Y 368.934,Z 184.03,A -85,B 0,C 180,E1 -12745.146,E2 -12745.146} C_VEL
LIN {X 0,Y 368.927,Z 184.028,A -85,B 0,C 180,E1 -12749.046,E2 -12749.046} C_VEL
LIN {X 0,Y 368.96,Z 184.025,A -85,B 0,C 180,E1 -12752.796,E2 -12752.796} C_VEL
LIN {X 0,Y 368.942,Z 184.028,A -85,B 0,C 180,E1 -12756.112,E2 -12756.112} C_VEL
LIN {X 0,Y 368.933,Z 184.028,A -85,B 0,C 180,E1 -12759.946,E2 -12759.946} C_VEL
LIN {X 0,Y 368.972,Z 184.021,A -85,B 0,C 180,E1 -12763.398,E2 -12763.398} C_VEL
LIN {X 0,Y 369.054,Z 184.011,A -85,B 0,C 180,E1 -12766.789,E2 -12766.789} C_VEL
LIN {X 0,Y 369.063,Z 184.014,A -85,B 0,C 180,E1 -12770.131,E2 -12770.131} C_VEL
LIN {X 0,Y 369.194,Z 183.995,A -85,B 0,C 180,E1 -12773.441,E2 -12773.441} C_VEL
LIN {X 0,Y 369.311,Z 183.984,A -85,B 0,C 180,E1 -12777.818,E2 -12777.818} C_VEL
LIN {X 0,Y 369.453,Z 183.964,A -85,B 0,C 180,E1 -12779.999,E2 -12779.999} C_VEL
LIN {X 0,Y 369.311,Z 183.98,A -85,B 0,C 180,E1 -12782.181,E2 -12782.181} C_VEL
LIN {X 0,Y 369.191,Z 183.993,A -85,B 0,C 180,E1 -12786.609,E2 -12786.609} C_VEL
LIN {X 0,Y 369.062,Z 184.011,A -85,B 0,C 180,E1 -12789.868,E2 -12789.868} C_VEL
LIN {X 0,Y 369.031,Z 184.015,A -85,B 0,C 180,E1 -12793.772,E2 -12793.772} C_VEL
LIN {X 0,Y 368.995,Z 184.019,A -85,B 0,C 180,E1 -12797.768,E2 -12797.768} C_VEL
LIN {X 0,Y 368.923,Z 184.031,A -85,B 0,C 180,E1 -12801.219,E2 -12801.219} C_VEL
LIN {X 0,Y 368.951,Z 184.028,A -85,B 0,C 180,E1 -12804.775,E2 -12804.775} C_VEL
LIN {X 0,Y 368.981,Z 184.022,A -85,B 0,C 180,E1 -12808.435,E2 -12808.435} C_VEL
LIN {X 0,Y 368.893,Z 184.032,A -85,B 0,C 180,E1 -12812.238,E2 -12812.238} C_VEL
LIN {X 0,Y 368.923,Z 184.03,A -85,B 0,C 180,E1 -12815.001,E2 -12815.001} C_VEL
LIN {X 0,Y 368.908,Z 184.034,A -85,B 0,C 180,E1 -12818.641,E2 -12818.641} C_VEL
LIN {X 0,Y 368.904,Z 184.03,A -85,B 0,C 180,E1 -12821.819,E2 -12821.819} C_VEL
LIN {X 0,Y 368.874,Z 184.033,A -85,B 0,C 180,E1 -12825.176,E2 -12825.176} C_VEL
LIN {X 0,Y 368.878,Z 184.038,A -85,B 0,C 180,E1 -12828.178,E2 -12828.178} C_VEL
LIN {X 0,Y 368.905,Z 184.029,A -85,B 0,C 180,E1 -12831.359,E2 -12831.359} C_VEL
LIN {X 0,Y 368.932,Z 184.026,A -85,B 0,C 180,E1 -12835.147,E2 -12835.147} C_VEL
LIN {X 0,Y 368.924,Z 184.027,A -85,B 0,C 180,E1 -12839.047,E2 -12839.047} C_VEL
LIN {X 0,Y 368.982,Z 184.023,A -85,B 0,C 180,E1 -12841.565,E2 -12841.565} C_VEL
LIN {X 0,Y 368.953,Z 184.025,A -85,B 0,C 180,E1 -12845.225,E2 -12845.225} C_VEL
LIN {X 0,Y 368.933,Z 184.026,A -85,B 0,C 180,E1 -12848.973,E2 -12848.973} C_VEL
LIN {X 0,Y 368.986,Z 184.024,A -85,B 0,C 180,E1 -12852.257,E2 -12852.257} C_VEL
LIN {X 0,Y 369.007,Z 184.079,A -85,B 0,C 180,E1 -12855.419,E2 -12855.419} C_VEL
LIN {X 0,Y 369.856,Z 186.616,A -85,B 0,C 180,E1 -12855.717,E2 -12855.717} C_VEL
LIN {X 0,Y 371.768,Z 188.778,A -85,B 0,C 180,E1 -12856.311,E2 -12856.311} C_VEL
LIN {X 0,Y 373.752,Z 190.11,A -85,B 0,C 180,E1 -12856.913,E2 -12856.913} C_VEL
LIN {X 0,Y 375.51,Z 193.026,A -85,B 0,C 180,E1 -12857.536,E2 -12857.536} C_VEL
LIN {X 0,Y 378.021,Z 195.221,A -85,B 0,C 180,E1 -12858.419,E2 -12858.419} C_VEL
LIN {X 0,Y 379.349,Z 196.066,A -85,B 0,C 180,E1 -12858.896,E2 -12858.896} C_VEL
LIN {X 0,Y 381.257,Z 198.944,A -85,B 0,C 180,E1 -12859.713,E2 -12859.713} C_VEL
LIN {X 0,Y 384.014,Z 201.231,A -85,B 0,C 180,E1 -12860.918,E2 -12860.918} C_VEL
LIN {X 0,Y 386.041,Z 202.341,A -85,B 0,C 180,E1 -12861.883,E2 -12861.883} C_VEL
LIN {X 0,Y 387.777,Z 204.96,A -85,B 0,C 180,E1 -12862.928,E2 -12862.928} C_VEL
LIN {X 0,Y 389.811,Z 207.005,A -85,B 0,C 180,E1 -12864.309,E2 -12864.309} C_VEL
LIN {X 0,Y 391.644,Z 208.136,A -85,B 0,C 180,E1 -12865.884,E2 -12865.884} C_VEL
LIN {X 0,Y 393.22,Z 208.524,A -85,B 0,C 180,E1 -12867.952,E2 -12867.952} C_VEL
LIN {X 0,Y 393.637,Z 208.55,A -85,B 0,C 180,E1 -12868.977,E2 -12868.977} C_VEL
LIN {X 0,Y 393.779,Z 208.579,A -85,B 0,C 180,E1 -12870,E2 -12870} C_VEL
LIN {X 0,Y 393.631,Z 208.552,A -85,B 0,C 180,E1 -12871.061,E2 -12871.061} C_VEL
LIN {X 0,Y 392.568,Z 208.349,A -85,B 0,C 180,E1 -12873.079,E2 -12873.079} C_VEL
LIN {X 0,Y 391.09,Z 207.883,A -85,B 0,C 180,E1 -12874.638,E2 -12874.638} C_VEL
LIN {X 0,Y 388.9,Z 206.243,A -85,B 0,C 180,E1 -12876.322,E2 -12876.322} C_VEL
LIN {X 0,Y 386.852,Z 203.725,A -85,B 0,C 180,E1 -12877.627,E2 -12877.627} C_VEL
LIN {X 0,Y 385.901,Z 202.054,A -85,B 0,C 180,E1 -12878.206,E2 -12878.206} C_VEL
LIN {X 0,Y 383.076,Z 200.611,A -85,B 0,C 180,E1 -12879.504,E2 -12879.504} C_VEL
LIN {X 0,Y 380.566,Z 198.105,A -85,B 0,C 180,E1 -12880.575,E2 -12880.575} C_VEL
LIN {X 0,Y 379.094,Z 195.76,A -85,B 0,C 180,E1 -12881.204,E2 -12881.204} C_VEL
LIN {X 0,Y 376.337,Z 193.947,A -85,B 0,C 180,E1 -12882.162,E2 -12882.162} C_VEL
LIN {X 0,Y 374.318,Z 191.247,A -85,B 0,C 180,E1 -12882.888,E2 -12882.888} C_VEL
LIN {X 0,Y 373.606,Z 189.801,A -85,B 0,C 180,E1 -12883.139,E2 -12883.139} C_VEL
LIN {X 0,Y 370.881,Z 187.991,A -85,B 0,C 180,E1 -12883.966,E2 -12883.966} C_VEL
LIN {X 0,Y 369.476,Z 185.837,A -85,B 0,C 180,E1 -12884.404,E2 -12884.404} C_VEL
LIN {X 0,Y 369.016,Z 184.022,A -85,B 0,C 180,E1 -12884.616,E2 -12884.616} C_VEL
LIN {X 0,Y 368.997,Z 184.022,A -85,B 0,C 180,E1 -12887.768,E2 -12887.768} C_VEL
LIN {X 0,Y 368.925,Z 184.027,A -85,B 0,C 180,E1 -12891.22,E2 -12891.22} C_VEL
LIN {X 0,Y 368.953,Z 184.025,A -85,B 0,C 180,E1 -12894.775,E2 -12894.775} C_VEL
LIN {X 0,Y 368.982,Z 184.023,A -85,B 0,C 180,E1 -12898.435,E2 -12898.435} C_VEL
LIN {X 0,Y 368.905,Z 184.033,A -85,B 0,C 180,E1 -12902.237,E2 -12902.237} C_VEL
LIN {X 0,Y 368.924,Z 184.027,A -85,B 0,C 180,E1 -12905.002,E2 -12905.002} C_VEL
LIN {X 0,Y 368.907,Z 184.029,A -85,B 0,C 180,E1 -12908.641,E2 -12908.641} C_VEL
LIN {X 0,Y 368.905,Z 184.035,A -85,B 0,C 180,E1 -12911.819,E2 -12911.819} C_VEL
LIN {X 0,Y 368.871,Z 184.033,A -85,B 0,C 180,E1 -12914.765,E2 -12914.765} C_VEL
LIN {X 0,Y 368.242,Z 184.118,A -85,B 0,C 180,E1 -12915.677,E2 -12915.677} C_VEL
LIN {X 0,Y 365.404,Z 184.471,A -85,B 0,C 180,E1 -12917.159,E2 -12917.159} C_VEL
LIN {X 0,Y 362.98,Z 184.772,A -85,B 0,C 180,E1 -12918.357,E2 -12918.357} C_VEL
LIN {X 0,Y 361.941,Z 184.9,A -85,B 0,C 180,E1 -12919.284,E2 -12919.284} C_VEL
LIN {X 0,Y 361.859,Z 184.908,A -85,B 0,C 180,E1 -12919.598,E2 -12919.598} C_VEL
LIN {X 0,Y 361.863,Z 184.908,A -85,B 0,C 180,E1 -12922.982,E2 -12922.982} C_VEL
LIN {X 0,Y 361.853,Z 184.908,A -85,B 0,C 180,E1 -12926.631,E2 -12926.631} C_VEL
LIN {X 0,Y 361.87,Z 184.907,A -85,B 0,C 180,E1 -12929.672,E2 -12929.672} C_VEL
LIN {X 0,Y 361.949,Z 184.898,A -85,B 0,C 180,E1 -12933.475,E2 -12933.475} C_VEL
LIN {X 0,Y 361.884,Z 184.908,A -85,B 0,C 180,E1 -12937.145,E2 -12937.145} C_VEL
LIN {X 0,Y 361.901,Z 184.906,A -85,B 0,C 180,E1 -12940.724,E2 -12940.724} C_VEL
LIN {X 0,Y 361.927,Z 184.902,A -85,B 0,C 180,E1 -12943.066,E2 -12943.066} C_VEL
LIN {X 0,Y 361.993,Z 184.894,A -85,B 0,C 180,E1 -12946.528,E2 -12946.528} C_VEL
LIN {X 0,Y 362.026,Z 184.887,A -85,B 0,C 180,E1 -12949.938,E2 -12949.938} C_VEL
LIN {X 0,Y 362.157,Z 184.87,A -85,B 0,C 180,E1 -12953.314,E2 -12953.314} C_VEL
LIN {X 0,Y 362.275,Z 184.856,A -85,B 0,C 180,E1 -12957.777,E2 -12957.777} C_VEL
LIN {X 0,Y 362.422,Z 184.84,A -85,B 0,C 180,E1 -12960.001,E2 -12960.001} C_VEL
LIN {X 0,Y 362.275,Z 184.861,A -85,B 0,C 180,E1 -12962.224,E2 -12962.224} C_VEL
LIN {X 0,Y 362.156,Z 184.871,A -85,B 0,C 180,E1 -12966.687,E2 -12966.687} C_VEL
LIN {X 0,Y 362.027,Z 184.892,A -85,B 0,C 180,E1 -12970.063,E2 -12970.063} C_VEL
LIN {X 0,Y 361.994,Z 184.896,A -85,B 0,C 180,E1 -12973.899,E2 -12973.899} C_VEL
LIN {X 0,Y 361.964,Z 184.898,A -85,B 0,C 180,E1 -12977.939,E2 -12977.939} C_VEL
LIN {X 0,Y 361.889,Z 184.909,A -85,B 0,C 180,E1 -12981.654,E2 -12981.654} C_VEL
LIN {X 0,Y 361.926,Z 184.902,A -85,B 0,C 180,E1 -12985.291,E2 -12985.291} C_VEL
LIN {X 0,Y 361.906,Z 184.904,A -85,B 0,C 180,E1 -12987.78,E2 -12987.78} C_VEL
LIN {X 0,Y 361.836,Z 184.913,A -85,B 0,C 180,E1 -12991.63,E2 -12991.63} C_VEL
LIN {X 0,Y 361.872,Z 184.911,A -85,B 0,C 180,E1 -12995.346,E2 -12995.346} C_VEL
LIN {X 0,Y 361.898,Z 185.117,A -85,B 0,C 180,E1 -12997.231,E2 -12997.231} C_VEL
LIN {X 0,Y 362.335,Z 188.039,A -85,B 0,C 180,E1 -13000.848,E2 -13000.848} C_VEL
LIN {X 0,Y 362.759,Z 191.038,A -85,B 0,C 180,E1 -13004.224,E2 -13004.224} C_VEL
LIN {X 0,Y 363.083,Z 194.096,A -85,B 0,C 180,E1 -13007.354,E2 -13007.354} C_VEL
LIN {X 0,Y 362.947,Z 197.203,A -85,B 0,C 180,E1 -13010.283,E2 -13010.283} C_VEL
LIN {X 0,Y 362.548,Z 200.366,A -85,B 0,C 180,E1 -13013.064,E2 -13013.064} C_VEL
LIN {X 0,Y 362.044,Z 204.604,A -85,B 0,C 180,E1 -13016.587,E2 -13016.587} C_VEL
LIN {X 0,Y 361.655,Z 208.464,A -85,B 0,C 180,E1 -13019.652,E2 -13019.652} C_VEL
LIN {X 0,Y 361.247,Z 213.43,A -85,B 0,C 180,E1 -13023.42,E2 -13023.42} C_VEL
LIN {X 0,Y 360.904,Z 218.436,A -85,B 0,C 180,E1 -13027.079,E2 -13027.079} C_VEL
LIN {X 0,Y 360.717,Z 222.55,A -85,B 0,C 180,E1 -13029.944,E2 -13029.944} C_VEL
LIN {X 0,Y 362.935,Z 232.989,A -85,B 0,C 180,E1 -13030.437,E2 -13030.437} C_VEL
LIN {X 0,Y 364.661,Z 242.466,A -85,B 0,C 180,E1 -13030.998,E2 -13030.998} C_VEL
LIN {X 0,Y 366.056,Z 252.218,A -85,B 0,C 180,E1 -13031.692,E2 -13031.692} C_VEL
LIN {X 0,Y 366.756,Z 257.911,A -85,B 0,C 180,E1 -13032.146,E2 -13032.146} C_VEL
LIN {X 0,Y 365.713,Z 268.823,A -85,B 0,C 180,E1 -13033.103,E2 -13033.103} C_VEL
LIN {X 0,Y 364.856,Z 277.772,A -85,B 0,C 180,E1 -13034.069,E2 -13034.069} C_VEL
LIN {X 0,Y 364.156,Z 284.826,A -85,B 0,C 180,E1 -13034.964,E2 -13034.964} C_VEL
LIN {X 0,Y 363.296,Z 293.53,A -85,B 0,C 180,E1 -13036.292,E2 -13036.292} C_VEL
LIN {X 0,Y 362.571,Z 299.734,A -85,B 0,C 180,E1 -13037.405,E2 -13037.405} C_VEL
LIN {X 0,Y 361.809,Z 306.272,A -85,B 0,C 180,E1 -13038.8,E2 -13038.8} C_VEL
LIN {X 0,Y 361.38,Z 310.777,A -85,B 0,C 180,E1 -13039.92,E2 -13039.92} C_VEL
LIN {X 0,Y 360.853,Z 316.271,A -85,B 0,C 180,E1 -13041.601,E2 -13041.601} C_VEL
LIN {X 0,Y 360.576,Z 320.6,A -85,B 0,C 180,E1 -13043.284,E2 -13043.284} C_VEL
LIN {X 0,Y 360.425,Z 322.967,A -85,B 0,C 180,E1 -13044.405,E2 -13044.405} C_VEL
LIN {X 0,Y 360.386,Z 324.768,A -85,B 0,C 180,E1 -13045.526,E2 -13045.526} C_VEL
LIN {X 0,Y 360.264,Z 327.213,A -85,B 0,C 180,E1 -13047.764,E2 -13047.764} C_VEL
LIN {X 0,Y 360.293,Z 327.803,A -85,B 0,C 180,E1 -13048.882,E2 -13048.882} C_VEL
LIN {X 0,Y 360.293,Z 327.803,A -85,B 0,C 180,E1 -13051.118,E2 -13051.118} C_VEL
LIN {X 0,Y 360.264,Z 327.213,A -85,B 0,C 180,E1 -13052.236,E2 -13052.236} C_VEL
LIN {X 0,Y 360.387,Z 324.768,A -85,B 0,C 180,E1 -13054.474,E2 -13054.474} C_VEL
LIN {X 0,Y 360.46,Z 321.974,A -85,B 0,C 180,E1 -13056.083,E2 -13056.083} C_VEL
LIN {X 0,Y 360.729,Z 317.826,A -85,B 0,C 180,E1 -13057.838,E2 -13057.838} C_VEL
LIN {X 0,Y 361.183,Z 312.694,A -85,B 0,C 180,E1 -13059.52,E2 -13059.52} C_VEL
LIN {X 0,Y 361.717,Z 307.429,A -85,B 0,C 180,E1 -13060.92,E2 -13060.92} C_VEL
LIN {X 0,Y 362.387,Z 301.109,A -85,B 0,C 180,E1 -13062.317,E2 -13062.317} C_VEL
LIN {X 0,Y 363.092,Z 295.157,A -85,B 0,C 180,E1 -13063.431,E2 -13063.431} C_VEL
LIN {X 0,Y 363.804,Z 288.226,A -85,B 0,C 180,E1 -13064.544,E2 -13064.544} C_VEL
LIN {X 0,Y 364.576,Z 280.041,A -85,B 0,C 180,E1 -13065.657,E2 -13065.657} C_VEL
LIN {X 0,Y 365.46,Z 271.527,A -85,B 0,C 180,E1 -13066.622,E2 -13066.622} C_VEL
LIN {X 0,Y 366.305,Z 262.81,A -85,B 0,C 180,E1 -13067.444,E2 -13067.444} C_VEL
LIN {X 0,Y 366.63,Z 256.877,A -85,B 0,C 180,E1 -13067.945,E2 -13067.945} C_VEL
LIN {X 0,Y 365,Z 244.591,A -85,B 0,C 180,E1 -13068.864,E2 -13068.864} C_VEL
LIN {X 0,Y 363.054,Z 233.683,A -85,B 0,C 180,E1 -13069.527,E2 -13069.527} C_VEL
LIN {X 0,Y 360.823,Z 223.401,A -85,B 0,C 180,E1 -13070.026,E2 -13070.026} C_VEL
LIN {X 0,Y 360.708,Z 222.389,A -85,B 0,C 180,E1 -13070.084,E2 -13070.084} C_VEL
LIN {X 0,Y 361.005,Z 216.746,A -85,B 0,C 180,E1 -13074.131,E2 -13074.131} C_VEL
LIN {X 0,Y 361.382,Z 211.759,A -85,B 0,C 180,E1 -13077.822,E2 -13077.822} C_VEL
LIN {X 0,Y 361.814,Z 206.824,A -85,B 0,C 180,E1 -13081.631,E2 -13081.631} C_VEL
LIN {X 0,Y 362.331,Z 202.138,A -85,B 0,C 180,E1 -13085.445,E2 -13085.445} C_VEL
LIN {X 0,Y 362.757,Z 198.775,A -85,B 0,C 180,E1 -13088.313,E2 -13088.313} C_VEL
LIN {X 0,Y 363.079,Z 195.624,A -85,B 0,C 180,E1 -13091.156,E2 -13091.156} C_VEL
LIN {X 0,Y 363.083,Z 194.062,A -85,B 0,C 180,E1 -13092.646,E2 -13092.646} C_VEL
LIN {X 0,Y 362.756,Z 191.018,A -85,B 0,C 180,E1 -13095.793,E2 -13095.793} C_VEL
LIN {X 0,Y 362.328,Z 188.02,A -85,B 0,C 180,E1 -13099.153,E2 -13099.153} C_VEL
LIN {X 0,Y 361.892,Z 185.122,A -85,B 0,C 180,E1 -13102.77,E2 -13102.77} C_VEL
LIN {X 0,Y 361.852,Z 184.913,A -85,B 0,C 180,E1 -13105.719,E2 -13105.719} C_VEL
LIN {X 0,Y 361.871,Z 184.905,A -85,B 0,C 180,E1 -13109.671,E2 -13109.671} C_VEL
LIN {X 0,Y 361.951,Z 184.895,A -85,B 0,C 180,E1 -13113.474,E2 -13113.474} C_VEL
LIN {X 0,Y 361.887,Z 184.904,A -85,B 0,C 180,E1 -13117.144,E2 -13117.144} C_VEL
LIN {X 0,Y 361.903,Z 184.903,A -85,B 0,C 180,E1 -13120.723,E2 -13120.723} C_VEL
LIN {X 0,Y 361.929,Z 184.898,A -85,B 0,C 180,E1 -13123.065,E2 -13123.065} C_VEL
LIN {X 0,Y 361.995,Z 184.892,A -85,B 0,C 180,E1 -13126.527,E2 -13126.527} C_VEL
LIN {X 0,Y 362.027,Z 184.892,A -85,B 0,C 180,E1 -13129.937,E2 -13129.937} C_VEL
LIN {X 0,Y 362.156,Z 184.871,A -85,B 0,C 180,E1 -13133.313,E2 -13133.313} C_VEL
LIN {X 0,Y 362.275,Z 184.861,A -85,B 0,C 180,E1 -13137.776,E2 -13137.776} C_VEL
LIN {X 0,Y 362.422,Z 184.84,A -85,B 0,C 180,E1 -13139.999,E2 -13139.999} C_VEL
LIN {X 0,Y 362.275,Z 184.856,A -85,B 0,C 180,E1 -13142.223,E2 -13142.223} C_VEL
LIN {X 0,Y 362.157,Z 184.87,A -85,B 0,C 180,E1 -13146.686,E2 -13146.686} C_VEL
LIN {X 0,Y 362.026,Z 184.887,A -85,B 0,C 180,E1 -13150.062,E2 -13150.062} C_VEL
LIN {X 0,Y 361.992,Z 184.891,A -85,B 0,C 180,E1 -13153.898,E2 -13153.898} C_VEL
LIN {X 0,Y 361.962,Z 184.894,A -85,B 0,C 180,E1 -13157.938,E2 -13157.938} C_VEL
LIN {X 0,Y 361.886,Z 184.904,A -85,B 0,C 180,E1 -13161.653,E2 -13161.653} C_VEL
LIN {X 0,Y 361.922,Z 184.902,A -85,B 0,C 180,E1 -13165.29,E2 -13165.29} C_VEL
LIN {X 0,Y 361.917,Z 184.9,A -85,B 0,C 180,E1 -13167.778,E2 -13167.778} C_VEL
LIN {X 0,Y 361.841,Z 184.911,A -85,B 0,C 180,E1 -13171.285,E2 -13171.285} C_VEL
LIN {X 0,Y 361.848,Z 184.911,A -85,B 0,C 180,E1 -13174.28,E2 -13174.28} C_VEL
LIN {X 0,Y 361.86,Z 184.908,A -85,B 0,C 180,E1 -13177.223,E2 -13177.223} C_VEL
LIN {X 0,Y 361.867,Z 184.909,A -85,B 0,C 180,E1 -13180.762,E2 -13180.762} C_VEL
LIN {X 0,Y 361.816,Z 184.919,A -85,B 0,C 180,E1 -13184.368,E2 -13184.368} C_VEL
LIN {X 0,Y 361.831,Z 184.911,A -85,B 0,C 180,E1 -13187.568,E2 -13187.568} C_VEL
LIN {X 0,Y 361.865,Z 184.906,A -85,B 0,C 180,E1 -13190.973,E2 -13190.973} C_VEL
LIN {X 0,Y 361.869,Z 184.907,A -85,B 0,C 180,E1 -13194.655,E2 -13194.655} C_VEL
LIN {X 0,Y 361.855,Z 184.91,A -85,B 0,C 180,E1 -13198.373,E2 -13198.373} C_VEL
LIN {X 0,Y 361.918,Z 184.902,A -85,B 0,C 180,E1 -13202.222,E2 -13202.222} C_VEL
LIN {X 0,Y 361.924,Z 184.899,A -85,B 0,C 180,E1 -13204.71,E2 -13204.71} C_VEL
LIN {X 0,Y 361.888,Z 184.904,A -85,B 0,C 180,E1 -13208.347,E2 -13208.347} C_VEL
LIN {X 0,Y 361.963,Z 184.898,A -85,B 0,C 180,E1 -13212.062,E2 -13212.062} C_VEL
LIN {X 0,Y 361.932,Z 184.903,A -85,B 0,C 180,E1 -13213.756,E2 -13213.756} C_VEL
LIN {X 0,Y 362.87,Z 187.66,A -85,B 0,C 180,E1 -13214.083,E2 -13214.083} C_VEL
LIN {X 0,Y 364.91,Z 189.822,A -85,B 0,C 180,E1 -13214.616,E2 -13214.616} C_VEL
LIN {X 0,Y 366.274,Z 190.777,A -85,B 0,C 180,E1 -13214.978,E2 -13214.978} C_VEL
LIN {X 0,Y 368.042,Z 193.678,A -85,B 0,C 180,E1 -13215.521,E2 -13215.521} C_VEL
LIN {X 0,Y 370.628,Z 195.881,A -85,B 0,C 180,E1 -13216.268,E2 -13216.268} C_VEL
LIN {X 0,Y 371.686,Z 196.935,A -85,B 0,C 180,E1 -13216.605,E2 -13216.605} C_VEL
LIN {X 0,Y 374.01,Z 200.044,A -85,B 0,C 180,E1 -13217.38,E2 -13217.38} C_VEL
LIN {X 0,Y 376.774,Z 202.182,A -85,B 0,C 180,E1 -13218.325,E2 -13218.325} C_VEL
LIN {X 0,Y 377.633,Z 202.921,A -85,B 0,C 180,E1 -13218.626,E2 -13218.626} C_VEL
LIN {X 0,Y 379.867,Z 205.849,A -85,B 0,C 180,E1 -13219.541,E2 -13219.541} C_VEL
LIN {X 0,Y 382.714,Z 208.12,A -85,B 0,C 180,E1 -13220.747,E2 -13220.747} C_VEL
LIN {X 0,Y 384.657,Z 209.162,A -85,B 0,C 180,E1 -13221.638,E2 -13221.638} C_VEL
LIN {X 0,Y 386.747,Z 212.039,A -85,B 0,C 180,E1 -13222.854,E2 -13222.854} C_VEL
LIN {X 0,Y 388.599,Z 213.878,A -85,B 0,C 180,E1 -13224.093,E2 -13224.093} C_VEL
LIN {X 0,Y 390.485,Z 215.074,A -85,B 0,C 180,E1 -13225.613,E2 -13225.613} C_VEL
LIN {X 0,Y 391.691,Z 215.396,A -85,B 0,C 180,E1 -13226.914,E2 -13226.914} C_VEL
LIN {X 0,Y 392.776,Z 215.597,A -85,B 0,C 180,E1 -13228.975,E2 -13228.975} C_VEL
LIN {X 0,Y 392.914,Z 215.625,A -85,B 0,C 180,E1 -13230,E2 -13230} C_VEL
LIN {X 0,Y 392.78,Z 215.572,A -85,B 0,C 180,E1 -13231.025,E2 -13231.025} C_VEL
LIN {X 0,Y 391.691,Z 215.394,A -85,B 0,C 180,E1 -13233.086,E2 -13233.086} C_VEL
LIN {X 0,Y 390.205,Z 214.909,A -85,B 0,C 180,E1 -13234.649,E2 -13234.649} C_VEL
LIN {X 0,Y 387.986,Z 213.359,A -85,B 0,C 180,E1 -13236.337,E2 -13236.337} C_VEL
LIN {X 0,Y 385.689,Z 210.76,A -85,B 0,C 180,E1 -13237.758,E2 -13237.758} C_VEL
LIN {X 0,Y 384.279,Z 208.826,A -85,B 0,C 180,E1 -13238.545,E2 -13238.545} C_VEL
LIN {X 0,Y 381.552,Z 207.292,A -85,B 0,C 180,E1 -13239.767,E2 -13239.767} C_VEL
LIN {X 0,Y 378.79,Z 204.621,A -85,B 0,C 180,E1 -13240.903,E2 -13240.903} C_VEL
LIN {X 0,Y 377.317,Z 202.477,A -85,B 0,C 180,E1 -13241.494,E2 -13241.494} C_VEL
LIN {X 0,Y 374.12,Z 200.147,A -85,B 0,C 180,E1 -13242.583,E2 -13242.583} C_VEL
LIN {X 0,Y 371.762,Z 197.068,A -85,B 0,C 180,E1 -13243.369,E2 -13243.369} C_VEL
LIN {X 0,Y 370.87,Z 196.028,A -85,B 0,C 180,E1 -13243.658,E2 -13243.658} C_VEL
LIN {X 0,Y 368.153,Z 193.834,A -85,B 0,C 180,E1 -13244.447,E2 -13244.447} C_VEL
LIN {X 0,Y 366.312,Z 190.867,A -85,B 0,C 180,E1 -13245.009,E2 -13245.009} C_VEL
LIN {X 0,Y 363.299,Z 188.292,A -85,B 0,C 180,E1 -13245.8,E2 -13245.8} C_VEL
LIN {X 0,Y 362.124,Z 185.85,A -85,B 0,C 180,E1 -13246.145,E2 -13246.145} C_VEL
LIN {X 0,Y 361.932,Z 184.903,A -85,B 0,C 180,E1 -13246.244,E2 -13246.244} C_VEL
LIN {X 0,Y 361.918,Z 184.904,A -85,B 0,C 180,E1 -13249.276,E2 -13249.276} C_VEL
LIN {X 0,Y 361.886,Z 184.905,A -85,B 0,C 180,E1 -13252.855,E2 -13252.855} C_VEL
LIN {X 0,Y 361.938,Z 184.898,A -85,B 0,C 180,E1 -13256.722,E2 -13256.722} C_VEL
LIN {X 0,Y 361.872,Z 184.909,A -85,B 0,C 180,E1 -13260.328,E2 -13260.328} C_VEL
LIN {X 0,Y 361.851,Z 184.911,A -85,B 0,C 180,E1 -13264.28,E2 -13264.28} C_VEL
LIN {X 0,Y 361.867,Z 184.907,A -85,B 0,C 180,E1 -13267.225,E2 -13267.225} C_VEL
LIN {X 0,Y 361.867,Z 184.906,A -85,B 0,C 180,E1 -13270.762,E2 -13270.762} C_VEL
LIN {X 0,Y 361.816,Z 184.913,A -85,B 0,C 180,E1 -13274.368,E2 -13274.368} C_VEL
LIN {X 0,Y 361.85,Z 184.914,A -85,B 0,C 180,E1 -13277.565,E2 -13277.565} C_VEL
LIN {X 0,Y 361.859,Z 184.908,A -85,B 0,C 180,E1 -13279.598,E2 -13279.598} C_VEL
LIN {X 0,Y 361.201,Z 184.99,A -85,B 0,C 180,E1 -13280.527,E2 -13280.527} C_VEL
LIN {X 0,Y 358.358,Z 185.344,A -85,B 0,C 180,E1 -13282.037,E2 -13282.037} C_VEL
LIN {X 0,Y 355.941,Z 185.649,A -85,B 0,C 180,E1 -13283.259,E2 -13283.259} C_VEL
LIN {X 0,Y 354.897,Z 185.775,A -85,B 0,C 180,E1 -13284.204,E2 -13284.204} C_VEL
LIN {X 0,Y 354.808,Z 185.785,A -85,B 0,C 180,E1 -13284.524,E2 -13284.524} C_VEL
LIN {X 0,Y 354.781,Z 185.791,A -85,B 0,C 180,E1 -13287.667,E2 -13287.667} C_VEL
LIN {X 0,Y 354.863,Z 185.78,A -85,B 0,C 180,E1 -13290.622,E2 -13290.622} C_VEL
LIN {X 0,Y 354.893,Z 185.775,A -85,B 0,C 180,E1 -13294.173,E2 -13294.173} C_VEL
LIN {X 0,Y 354.829,Z 185.783,A -85,B 0,C 180,E1 -13297.894,E2 -13297.894} C_VEL
LIN {X 0,Y 354.917,Z 185.772,A -85,B 0,C 180,E1 -13301.892,E2 -13301.892} C_VEL
LIN {X 0,Y 354.937,Z 185.77,A -85,B 0,C 180,E1 -13305.982,E2 -13305.982} C_VEL
LIN {X 0,Y 354.972,Z 185.765,A -85,B 0,C 180,E1 -13309.736,E2 -13309.736} C_VEL
LIN {X 0,Y 355.121,Z 185.747,A -85,B 0,C 180,E1 -13313.181,E2 -13313.181} C_VEL
LIN {X 0,Y 355.238,Z 185.732,A -85,B 0,C 180,E1 -13317.733,E2 -13317.733} C_VEL
LIN {X 0,Y 355.392,Z 185.715,A -85,B 0,C 180,E1 -13320.001,E2 -13320.001} C_VEL
LIN {X 0,Y 355.238,Z 185.738,A -85,B 0,C 180,E1 -13322.268,E2 -13322.268} C_VEL
LIN {X 0,Y 355.119,Z 185.747,A -85,B 0,C 180,E1 -13326.82,E2 -13326.82} C_VEL
LIN {X 0,Y 354.974,Z 185.768,A -85,B 0,C 180,E1 -13330.265,E2 -13330.265} C_VEL
LIN {X 0,Y 354.939,Z 185.774,A -85,B 0,C 180,E1 -13334.019,E2 -13334.019} C_VEL
LIN {X 0,Y 354.919,Z 185.774,A -85,B 0,C 180,E1 -13338.109,E2 -13338.109} C_VEL
LIN {X 0,Y 354.832,Z 185.784,A -85,B 0,C 180,E1 -13342.107,E2 -13342.107} C_VEL
LIN {X 0,Y 354.896,Z 185.778,A -85,B 0,C 180,E1 -13345.828,E2 -13345.828} C_VEL
LIN {X 0,Y 354.815,Z 185.788,A -85,B 0,C 180,E1 -13349.683,E2 -13349.683} C_VEL
LIN {X 0,Y 354.804,Z 185.79,A -85,B 0,C 180,E1 -13353.703,E2 -13353.703} C_VEL
LIN {X 0,Y 354.797,Z 185.792,A -85,B 0,C 180,E1 -13356.46,E2 -13356.46} C_VEL
LIN {X 0,Y 355.152,Z 188.044,A -85,B 0,C 180,E1 -13359.489,E2 -13359.489} C_VEL
LIN {X 0,Y 355.582,Z 191.008,A -85,B 0,C 180,E1 -13363.006,E2 -13363.006} C_VEL
LIN {X 0,Y 355.95,Z 194.048,A -85,B 0,C 180,E1 -13366.287,E2 -13366.287} C_VEL
LIN {X 0,Y 356.004,Z 197.156,A -85,B 0,C 180,E1 -13369.349,E2 -13369.349} C_VEL
LIN {X 0,Y 355.625,Z 200.312,A -85,B 0,C 180,E1 -13372.233,E2 -13372.233} C_VEL
LIN {X 0,Y 355.214,Z 203.483,A -85,B 0,C 180,E1 -13374.987,E2 -13374.987} C_VEL
LIN {X 0,Y 354.684,Z 208.346,A -85,B 0,C 180,E1 -13378.991,E2 -13378.991} C_VEL
LIN {X 0,Y 354.366,Z 211.617,A -85,B 0,C 180,E1 -13381.577,E2 -13381.577} C_VEL
LIN {X 0,Y 354.073,Z 214.922,A -85,B 0,C 180,E1 -13384.108,E2 -13384.108} C_VEL
LIN {X 0,Y 353.876,Z 218.267,A -85,B 0,C 180,E1 -13386.597,E2 -13386.597} C_VEL
LIN {X 0,Y 353.665,Z 222.195,A -85,B 0,C 180,E1 -13389.517,E2 -13389.517} C_VEL
LIN {X 0,Y 356.04,Z 233.374,A -85,B 0,C 180,E1 -13390.069,E2 -13390.069} C_VEL
LIN {X 0,Y 357.86,Z 243.503,A -85,B 0,C 180,E1 -13390.695,E2 -13390.695} C_VEL
LIN {X 0,Y 359.382,Z 254.643,A -85,B 0,C 180,E1 -13391.532,E2 -13391.532} C_VEL
LIN {X 0,Y 359.854,Z 259.334,A -85,B 0,C 180,E1 -13391.939,E2 -13391.939} C_VEL
LIN {X 0,Y 358.915,Z 268.611,A -85,B 0,C 180,E1 -13392.773,E2 -13392.773} C_VEL
LIN {X 0,Y 357.983,Z 277.559,A -85,B 0,C 180,E1 -13393.754,E2 -13393.754} C_VEL
LIN {X 0,Y 357.193,Z 285.362,A -85,B 0,C 180,E1 -13394.777,E2 -13394.777} C_VEL
LIN {X 0,Y 356.356,Z 293.318,A -85,B 0,C 180,E1 -13396.02,E2 -13396.02} C_VEL
LIN {X 0,Y 355.609,Z 299.521,A -85,B 0,C 180,E1 -13397.154,E2 -13397.154} C_VEL
LIN {X 0,Y 354.801,Z 306.06,A -85,B 0,C 180,E1 -13398.575,E2 -13398.575} C_VEL
LIN {X 0,Y 354.358,Z 310.565,A -85,B 0,C 180,E1 -13399.718,E2 -13399.718} C_VEL
LIN {X 0,Y 353.816,Z 316.059,A -85,B 0,C 180,E1 -13401.433,E2 -13401.433} C_VEL
LIN {X 0,Y 353.509,Z 320.388,A -85,B 0,C 180,E1 -13403.149,E2 -13403.149} C_VEL
LIN {X 0,Y 353.332,Z 322.755,A -85,B 0,C 180,E1 -13404.292,E2 -13404.292} C_VEL
LIN {X 0,Y 353.3,Z 324.557,A -85,B 0,C 180,E1 -13405.436,E2 -13405.436} C_VEL
LIN {X 0,Y 353.172,Z 327.002,A -85,B 0,C 180,E1 -13407.719,E2 -13407.719} C_VEL
LIN {X 0,Y 353.194,Z 327.592,A -85,B 0,C 180,E1 -13408.86,E2 -13408.86} C_VEL
LIN {X 0,Y 353.194,Z 327.592,A -85,B 0,C 180,E1 -13411.14,E2 -13411.14} C_VEL
LIN {X 0,Y 353.172,Z 327.002,A -85,B 0,C 180,E1 -13412.281,E2 -13412.281} C_VEL
LIN {X 0,Y 353.3,Z 324.557,A -85,B 0,C 180,E1 -13414.564,E2 -13414.564} C_VEL
LIN {X 0,Y 353.371,Z 322.091,A -85,B 0,C 180,E1 -13416.051,E2 -13416.051} C_VEL
LIN {X 0,Y 353.549,Z 319.145,A -85,B 0,C 180,E1 -13417.424,E2 -13417.424} C_VEL
LIN {X 0,Y 353.979,Z 314.398,A -85,B 0,C 180,E1 -13419.139,E2 -13419.139} C_VEL
LIN {X 0,Y 354.613,Z 308.374,A -85,B 0,C 180,E1 -13420.852,E2 -13420.852} C_VEL
LIN {X 0,Y 355.238,Z 302.273,A -85,B 0,C 180,E1 -13422.279,E2 -13422.279} C_VEL
LIN {X 0,Y 355.968,Z 296.572,A -85,B 0,C 180,E1 -13423.414,E2 -13423.414} C_VEL
LIN {X 0,Y 356.92,Z 288.015,A -85,B 0,C 180,E1 -13424.831,E2 -13424.831} C_VEL
LIN {X 0,Y 357.721,Z 279.829,A -85,B 0,C 180,E1 -13425.965,E2 -13425.965} C_VEL
LIN {X 0,Y 358.643,Z 271.316,A -85,B 0,C 180,E1 -13426.947,E2 -13426.947} C_VEL
LIN {X 0,Y 359.533,Z 262.598,A -85,B 0,C 180,E1 -13427.784,E2 -13427.784} C_VEL
LIN {X 0,Y 359.725,Z 257.691,A -85,B 0,C 180,E1 -13428.215,E2 -13428.215} C_VEL
LIN {X 0,Y 358.242,Z 245.859,A -85,B 0,C 180,E1 -13429.148,E2 -13429.148} C_VEL
LIN {X 0,Y 356.159,Z 234.144,A -85,B 0,C 180,E1 -13429.892,E2 -13429.892} C_VEL
LIN {X 0,Y 353.838,Z 223.663,A -85,B 0,C 180,E1 -13430.425,E2 -13430.425} C_VEL
LIN {X 0,Y 353.658,Z 222.168,A -85,B 0,C 180,E1 -13430.502,E2 -13430.502} C_VEL
LIN {X 0,Y 353.954,Z 216.583,A -85,B 0,C 180,E1 -13434.643,E2 -13434.643} C_VEL
LIN {X 0,Y 354.232,Z 213.266,A -85,B 0,C 180,E1 -13437.15,E2 -13437.15} C_VEL
LIN {X 0,Y 354.498,Z 209.981,A -85,B 0,C 180,E1 -13439.711,E2 -13439.711} C_VEL
LIN {X 0,Y 354.838,Z 206.717,A -85,B 0,C 180,E1 -13442.328,E2 -13442.328} C_VEL
LIN {X 0,Y 355.335,Z 202.545,A -85,B 0,C 180,E1 -13445.813,E2 -13445.813} C_VEL
LIN {X 0,Y 355.906,Z 198.229,A -85,B 0,C 180,E1 -13449.634,E2 -13449.634} C_VEL
LIN {X 0,Y 356.023,Z 195.575,A -85,B 0,C 180,E1 -13452.157,E2 -13452.157} C_VEL
LIN {X 0,Y 355.762,Z 192.511,A -85,B 0,C 180,E1 -13455.329,E2 -13455.329} C_VEL
LIN {X 0,Y 355.384,Z 189.5,A -85,B 0,C 180,E1 -13458.718,E2 -13458.718} C_VEL
LIN {X 0,Y 354.915,Z 186.579,A -85,B 0,C 180,E1 -13462.379,E2 -13462.379} C_VEL
LIN {X 0,Y 354.794,Z 185.79,A -85,B 0,C 180,E1 -13463.539,E2 -13463.539} C_VEL
LIN {X 0,Y 354.812,Z 185.79,A -85,B 0,C 180,E1 -13466.315,E2 -13466.315} C_VEL
LIN {X 0,Y 354.815,Z 185.788,A -85,B 0,C 180,E1 -13470.317,E2 -13470.317} C_VEL
LIN {X 0,Y 354.896,Z 185.778,A -85,B 0,C 180,E1 -13474.172,E2 -13474.172} C_VEL
LIN {X 0,Y 354.832,Z 185.784,A -85,B 0,C 180,E1 -13477.893,E2 -13477.893} C_VEL
LIN {X 0,Y 354.919,Z 185.774,A -85,B 0,C 180,E1 -13481.891,E2 -13481.891} C_VEL
LIN {X 0,Y 354.939,Z 185.774,A -85,B 0,C 180,E1 -13485.981,E2 -13485.981} C_VEL
LIN {X 0,Y 354.974,Z 185.768,A -85,B 0,C 180,E1 -13489.735,E2 -13489.735} C_VEL
LIN {X 0,Y 355.119,Z 185.747,A -85,B 0,C 180,E1 -13493.18,E2 -13493.18} C_VEL
LIN {X 0,Y 355.238,Z 185.738,A -85,B 0,C 180,E1 -13497.732,E2 -13497.732} C_VEL
LIN {X 0,Y 355.392,Z 185.715,A -85,B 0,C 180,E1 -13499.999,E2 -13499.999} C_VEL
LIN {X 0,Y 355.238,Z 185.732,A -85,B 0,C 180,E1 -13502.267,E2 -13502.267} C_VEL
LIN {X 0,Y 355.121,Z 185.747,A -85,B 0,C 180,E1 -13506.819,E2 -13506.819} C_VEL
LIN {X 0,Y 354.972,Z 185.765,A -85,B 0,C 180,E1 -13510.264,E2 -13510.264} C_VEL
LIN {X 0,Y 354.937,Z 185.77,A -85,B 0,C 180,E1 -13514.018,E2 -13514.018} C_VEL
LIN {X 0,Y 354.917,Z 185.772,A -85,B 0,C 180,E1 -13518.108,E2 -13518.108} C_VEL
LIN {X 0,Y 354.829,Z 185.783,A -85,B 0,C 180,E1 -13522.106,E2 -13522.106} C_VEL
LIN {X 0,Y 354.893,Z 185.775,A -85,B 0,C 180,E1 -13525.827,E2 -13525.827} C_VEL
LIN {X 0,Y 354.849,Z 185.78,A -85,B 0,C 180,E1 -13529.678,E2 -13529.678} C_VEL
LIN {X 0,Y 354.8,Z 185.786,A -85,B 0,C 180,E1 -13533.702,E2 -13533.702} C_VEL
LIN {X 0,Y 354.794,Z 185.792,A -85,B 0,C 180,E1 -13536.459,E2 -13536.459} C_VEL
LIN {X 0,Y 354.818,Z 185.784,A -85,B 0,C 180,E1 -13539.423,E2 -13539.423} C_VEL
LIN {X 0,Y 354.798,Z 185.788,A -85,B 0,C 180,E1 -13542.87,E2 -13542.87} C_VEL
LIN {X 0,Y 354.762,Z 185.795,A -85,B 0,C 180,E1 -13546.104,E2 -13546.104} C_VEL
LIN {X 0,Y 354.783,Z 185.788,A -85,B 0,C 180,E1 -13549.179,E2 -13549.179} C_VEL
LIN {X 0,Y 354.803,Z 185.789,A -85,B 0,C 180,E1 -13552.402,E2 -13552.402} C_VEL
LIN {X 0,Y 354.807,Z 185.785,A -85,B 0,C 180,E1 -13554.941,E2 -13554.941} C_VEL
LIN {X 0,Y 354.81,Z 185.787,A -85,B 0,C 180,E1 -13558.399,E2 -13558.399} C_VEL
LIN {X 0,Y 354.849,Z 185.784,A -85,B 0,C 180,E1 -13561.619,E2 -13561.619} C_VEL
LIN {X 0,Y 354.895,Z 185.777,A -85,B 0,C 180,E1 -13564.173,E2 -13564.173} C_VEL
LIN {X 0,Y 354.831,Z 185.786,A -85,B 0,C 180,E1 -13567.894,E2 -13567.894} C_VEL
LIN {X 0,Y 354.919,Z 185.776,A -85,B 0,C 180,E1 -13571.891,E2 -13571.891} C_VEL
LIN {X 0,Y 354.913,Z 185.778,A -85,B 0,C 180,E1 -13572.332,E2 -13572.332} C_VEL
LIN {X 0,Y 355.753,Z 188.365,A -85,B 0,C 180,E1 -13572.588,E2 -13572.588} C_VEL
LIN {X 0,Y 357.644,Z 190.561,A -85,B 0,C 180,E1 -13573.045,E2 -13573.045} C_VEL
LIN {X 0,Y 358.962,Z 191.682,A -85,B 0,C 180,E1 -13573.351,E2 -13573.351} C_VEL
LIN {X 0,Y 360.857,Z 194.636,A -85,B 0,C 180,E1 -13573.864,E2 -13573.864} C_VEL
LIN {X 0,Y 363.789,Z 197.36,A -85,B 0,C 180,E1 -13574.619,E2 -13574.619} C_VEL
LIN {X 0,Y 366.328,Z 200.657,A -85,B 0,C 180,E1 -13575.345,E2 -13575.345} C_VEL
LIN {X 0,Y 369.355,Z 203.182,A -85,B 0,C 180,E1 -13576.202,E2 -13576.202} C_VEL
LIN {X 0,Y 372.187,Z 206.694,A -85,B 0,C 180,E1 -13577.118,E2 -13577.118} C_VEL
LIN {X 0,Y 375.801,Z 209.595,A -85,B 0,C 180,E1 -13578.336,E2 -13578.336} C_VEL
LIN {X 0,Y 378.294,Z 212.564,A -85,B 0,C 180,E1 -13579.293,E2 -13579.293} C_VEL
LIN {X 0,Y 381.408,Z 215.014,A -85,B 0,C 180,E1 -13580.584,E2 -13580.584} C_VEL
LIN {X 0,Y 383.282,Z 216.108,A -85,B 0,C 180,E1 -13581.432,E2 -13581.432} C_VEL
LIN {X 0,Y 385.714,Z 219.118,A -85,B 0,C 180,E1 -13582.781,E2 -13582.781} C_VEL
LIN {X 0,Y 387.686,Z 220.944,A -85,B 0,C 180,E1 -13584.079,E2 -13584.079} C_VEL
LIN {X 0,Y 389.596,Z 222.12,A -85,B 0,C 180,E1 -13585.603,E2 -13585.603} C_VEL
LIN {X 0,Y 390.814,Z 222.441,A -85,B 0,C 180,E1 -13586.908,E2 -13586.908} C_VEL
LIN {X 0,Y 391.493,Z 222.61,A -85,B 0,C 180,E1 -13587.942,E2 -13587.942} C_VEL
LIN {X 0,Y 391.912,Z 222.643,A -85,B 0,C 180,E1 -13588.972,E2 -13588.972} C_VEL
LIN {X 0,Y 392.049,Z 222.672,A -85,B 0,C 180,E1 -13590,E2 -13590} C_VEL
LIN {X 0,Y 391.916,Z 222.615,A -85,B 0,C 180,E1 -13591.027,E2 -13591.027} C_VEL
LIN {X 0,Y 391.493,Z 222.602,A -85,B 0,C 180,E1 -13592.058,E2 -13592.058} C_VEL
LIN {X 0,Y 389.866,Z 222.222,A -85,B 0,C 180,E1 -13594.135,E2 -13594.135} C_VEL
LIN {X 0,Y 387.986,Z 221.124,A -85,B 0,C 180,E1 -13595.718,E2 -13595.718} C_VEL
LIN {X 0,Y 385.835,Z 219.28,A -85,B 0,C 180,E1 -13597.14,E2 -13597.14} C_VEL
LIN {X 0,Y 383.282,Z 216.109,A -85,B 0,C 180,E1 -13598.568,E2 -13598.568} C_VEL
LIN {X 0,Y 379.719,Z 213.836,A -85,B 0,C 180,E1 -13600.127,E2 -13600.127} C_VEL
LIN {X 0,Y 376.75,Z 210.888,A -85,B 0,C 180,E1 -13601.31,E2 -13601.31} C_VEL
LIN {X 0,Y 375.166,Z 208.961,A -85,B 0,C 180,E1 -13601.892,E2 -13601.892} C_VEL
LIN {X 0,Y 372.031,Z 206.556,A -85,B 0,C 180,E1 -13602.93,E2 -13602.93} C_VEL
LIN {X 0,Y 369.213,Z 202.971,A -85,B 0,C 180,E1 -13603.842,E2 -13603.842} C_VEL
LIN {X 0,Y 365.598,Z 199.898,A -85,B 0,C 180,E1 -13604.863,E2 -13604.863} C_VEL
LIN {X 0,Y 363.096,Z 196.594,A -85,B 0,C 180,E1 -13605.563,E2 -13605.563} C_VEL
LIN {X 0,Y 360.46,Z 194.151,A -85,B 0,C 180,E1 -13606.242,E2 -13606.242} C_VEL
LIN {X 0,Y 358.64,Z 191.197,A -85,B 0,C 180,E1 -13606.73,E2 -13606.73} C_VEL
LIN {X 0,Y 356.271,Z 189.191,A -85,B 0,C 180,E1 -13607.28,E2 -13607.28} C_VEL
LIN {X 0,Y 355.063,Z 186.665,A -85,B 0,C 180,E1 -13607.608,E2 -13607.608} C_VEL
LIN {X 0,Y 354.921,Z 185.776,A -85,B 0,C 180,E1 -13607.693,E2 -13607.693} C_VEL
LIN {X 0,Y 354.837,Z 185.782,A -85,B 0,C 180,E1 -13611.427,E2 -13611.427} C_VEL
LIN {X 0,Y 354.857,Z 185.782,A -85,B 0,C 180,E1 -13614.576,E2 -13614.576} C_VEL
LIN {X 0,Y 354.88,Z 185.776,A -85,B 0,C 180,E1 -13617.096,E2 -13617.096} C_VEL
LIN {X 0,Y 354.85,Z 185.782,A -85,B 0,C 180,E1 -13619.678,E2 -13619.678} C_VEL
LIN {X 0,Y 354.826,Z 185.786,A -85,B 0,C 180,E1 -13623.682,E2 -13623.682} C_VEL
LIN {X 0,Y 354.797,Z 185.788,A -85,B 0,C 180,E1 -13626.459,E2 -13626.459} C_VEL
LIN {X 0,Y 354.819,Z 185.786,A -85,B 0,C 180,E1 -13629.424,E2 -13629.424} C_VEL
LIN {X 0,Y 354.799,Z 185.787,A -85,B 0,C 180,E1 -13632.87,E2 -13632.87} C_VEL
LIN {X 0,Y 354.798,Z 185.788,A -85,B 0,C 180,E1 -13637.13,E2 -13637.13} C_VEL
LIN {X 0,Y 354.832,Z 185.783,A -85,B 0,C 180,E1 -13640.669,E2 -13640.669} C_VEL
LIN {X 0,Y 354.808,Z 185.785,A -85,B 0,C 180,E1 -13644.524,E2 -13644.524} C_VEL
LIN {X 0,Y 354.118,Z 185.876,A -85,B 0,C 180,E1 -13645.471,E2 -13645.471} C_VEL
LIN {X 0,Y 351.222,Z 186.235,A -85,B 0,C 180,E1 -13647.011,E2 -13647.011} C_VEL
LIN {X 0,Y 348.806,Z 186.533,A -85,B 0,C 180,E1 -13648.257,E2 -13648.257} C_VEL
LIN {X 0,Y 347.81,Z 186.663,A -85,B 0,C 180,E1 -13649.222,E2 -13649.222} C_VEL
LIN {X 0,Y 347.75,Z 186.666,A -85,B 0,C 180,E1 -13649.548,E2 -13649.548} C_VEL
LIN {X 0,Y 347.847,Z 186.655,A -85,B 0,C 180,E1 -13652.745,E2 -13652.745} C_VEL
LIN {X 0,Y 347.783,Z 186.66,A -85,B 0,C 180,E1 -13656.162,E2 -13656.162} C_VEL
LIN {X 0,Y 347.807,Z 186.657,A -85,B 0,C 180,E1 -13659.91,E2 -13659.91} C_VEL
LIN {X 0,Y 347.86,Z 186.652,A -85,B 0,C 180,E1 -13662.36,E2 -13662.36} C_VEL
LIN {X 0,Y 347.892,Z 186.647,A -85,B 0,C 180,E1 -13665.971,E2 -13665.971} C_VEL
LIN {X 0,Y 347.923,Z 186.643,A -85,B 0,C 180,E1 -13669.526,E2 -13669.526} C_VEL
LIN {X 0,Y 348.087,Z 186.624,A -85,B 0,C 180,E1 -13673.043,E2 -13673.043} C_VEL
LIN {X 0,Y 348.201,Z 186.607,A -85,B 0,C 180,E1 -13677.687,E2 -13677.687} C_VEL
LIN {X 0,Y 348.341,Z 186.593,A -85,B 0,C 180,E1 -13680.001,E2 -13680.001} C_VEL
LIN {X 0,Y 348.2,Z 186.614,A -85,B 0,C 180,E1 -13682.314,E2 -13682.314} C_VEL
LIN {X 0,Y 348.086,Z 186.623,A -85,B 0,C 180,E1 -13686.959,E2 -13686.959} C_VEL
LIN {X 0,Y 347.924,Z 186.645,A -85,B 0,C 180,E1 -13690.475,E2 -13690.475} C_VEL
LIN {X 0,Y 347.895,Z 186.65,A -85,B 0,C 180,E1 -13694.151,E2 -13694.151} C_VEL
LIN {X 0,Y 347.887,Z 186.649,A -85,B 0,C 180,E1 -13698.291,E2 -13698.291} C_VEL
LIN {X 0,Y 347.786,Z 186.666,A -85,B 0,C 180,E1 -13701.636,E2 -13701.636} C_VEL
LIN {X 0,Y 347.81,Z 186.659,A -85,B 0,C 180,E1 -13705.109,E2 -13705.109} C_VEL
LIN {X 0,Y 347.806,Z 186.662,A -85,B 0,C 180,E1 -13707.695,E2 -13707.695} C_VEL
LIN {X 0,Y 347.747,Z 186.666,A -85,B 0,C 180,E1 -13710.349,E2 -13710.349} C_VEL
LIN {X 0,Y 347.746,Z 186.669,A -85,B 0,C 180,E1 -13714.045,E2 -13714.045} C_VEL
LIN {X 0,Y 347.769,Z 186.666,A -85,B 0,C 180,E1 -13716.066,E2 -13716.066} C_VEL
LIN {X 0,Y 348.21,Z 189.524,A -85,B 0,C 180,E1 -13719.919,E2 -13719.919} C_VEL
LIN {X 0,Y 348.638,Z 192.494,A -85,B 0,C 180,E1 -13723.473,E2 -13723.473} C_VEL
LIN {X 0,Y 348.951,Z 195.544,A -85,B 0,C 180,E1 -13726.783,E2 -13726.783} C_VEL
LIN {X 0,Y 348.904,Z 198.731,A -85,B 0,C 180,E1 -13729.947,E2 -13729.947} C_VEL
LIN {X 0,Y 348.347,Z 202.967,A -85,B 0,C 180,E1 -13733.806,E2 -13733.806} C_VEL
LIN {X 0,Y 347.864,Z 206.606,A -85,B 0,C 180,E1 -13736.943,E2 -13736.943} C_VEL
LIN {X 0,Y 347.433,Z 210.844,A -85,B 0,C 180,E1 -13740.439,E2 -13740.439} C_VEL
LIN {X 0,Y 347.079,Z 214.777,A -85,B 0,C 180,E1 -13743.547,E2 -13743.547} C_VEL
LIN {X 0,Y 346.839,Z 218.072,A -85,B 0,C 180,E1 -13746.093,E2 -13746.093} C_VEL
LIN {X 0,Y 346.593,Z 222.034,A -85,B 0,C 180,E1 -13749.088,E2 -13749.088} C_VEL
LIN {X 0,Y 348.799,Z 232.146,A -85,B 0,C 180,E1 -13749.593,E2 -13749.593} C_VEL
LIN {X 0,Y 350.595,Z 241.532,A -85,B 0,C 180,E1 -13750.176,E2 -13750.176} C_VEL
LIN {X 0,Y 351.94,Z 250.676,A -85,B 0,C 180,E1 -13750.847,E2 -13750.847} C_VEL
LIN {X 0,Y 352.933,Z 259.117,A -85,B 0,C 180,E1 -13751.572,E2 -13751.572} C_VEL
LIN {X 0,Y 352.128,Z 268.4,A -85,B 0,C 180,E1 -13752.43,E2 -13752.43} C_VEL
LIN {X 0,Y 351.133,Z 277.346,A -85,B 0,C 180,E1 -13753.428,E2 -13753.428} C_VEL
LIN {X 0,Y 350.224,Z 285.939,A -85,B 0,C 180,E1 -13754.589,E2 -13754.589} C_VEL
LIN {X 0,Y 349.422,Z 293.105,A -85,B 0,C 180,E1 -13755.736,E2 -13755.736} C_VEL
LIN {X 0,Y 348.642,Z 299.308,A -85,B 0,C 180,E1 -13756.893,E2 -13756.893} C_VEL
LIN {X 0,Y 347.805,Z 305.847,A -85,B 0,C 180,E1 -13758.342,E2 -13758.342} C_VEL
LIN {X 0,Y 347.353,Z 310.353,A -85,B 0,C 180,E1 -13759.508,E2 -13759.508} C_VEL
LIN {X 0,Y 346.763,Z 315.847,A -85,B 0,C 180,E1 -13761.257,E2 -13761.257} C_VEL
LIN {X 0,Y 346.422,Z 320.175,A -85,B 0,C 180,E1 -13763.008,E2 -13763.008} C_VEL
LIN {X 0,Y 346.251,Z 322.543,A -85,B 0,C 180,E1 -13764.175,E2 -13764.175} C_VEL
LIN {X 0,Y 346.216,Z 324.345,A -85,B 0,C 180,E1 -13765.343,E2 -13765.343} C_VEL
LIN {X 0,Y 346.084,Z 326.791,A -85,B 0,C 180,E1 -13767.672,E2 -13767.672} C_VEL
LIN {X 0,Y 346.095,Z 327.381,A -85,B 0,C 180,E1 -13768.836,E2 -13768.836} C_VEL
LIN {X 0,Y 346.095,Z 327.381,A -85,B 0,C 180,E1 -13771.164,E2 -13771.164} C_VEL
LIN {X 0,Y 346.084,Z 326.791,A -85,B 0,C 180,E1 -13772.328,E2 -13772.328} C_VEL
LIN {X 0,Y 346.216,Z 324.345,A -85,B 0,C 180,E1 -13774.657,E2 -13774.657} C_VEL
LIN {X 0,Y 346.345,Z 321.394,A -85,B 0,C 180,E1 -13776.407,E2 -13776.407} C_VEL
LIN {X 0,Y 346.617,Z 317.402,A -85,B 0,C 180,E1 -13778.16,E2 -13778.16} C_VEL
LIN {X 0,Y 347.116,Z 312.269,A -85,B 0,C 180,E1 -13779.91,E2 -13779.91} C_VEL
LIN {X 0,Y 347.697,Z 307.004,A -85,B 0,C 180,E1 -13781.366,E2 -13781.366} C_VEL
LIN {X 0,Y 348.459,Z 300.685,A -85,B 0,C 180,E1 -13782.818,E2 -13782.818} C_VEL
LIN {X 0,Y 349.209,Z 294.732,A -85,B 0,C 180,E1 -13783.975,E2 -13783.975} C_VEL
LIN {X 0,Y 350.149,Z 286.802,A -85,B 0,C 180,E1 -13785.28,E2 -13785.28} C_VEL
LIN {X 0,Y 350.859,Z 279.616,A -85,B 0,C 180,E1 -13786.286,E2 -13786.286} C_VEL
LIN {X 0,Y 351.822,Z 271.103,A -85,B 0,C 180,E1 -13787.286,E2 -13787.286} C_VEL
LIN {X 0,Y 352.774,Z 262.387,A -85,B 0,C 180,E1 -13788.136,E2 -13788.136} C_VEL
LIN {X 0,Y 352.759,Z 257.473,A -85,B 0,C 180,E1 -13788.588,E2 -13788.588} C_VEL
LIN {X 0,Y 351.297,Z 245.746,A -85,B 0,C 180,E1 -13789.536,E2 -13789.536} C_VEL
LIN {X 0,Y 349.213,Z 234.028,A -85,B 0,C 180,E1 -13790.3,E2 -13790.3} C_VEL
LIN {X 0,Y 346.771,Z 223.346,A -85,B 0,C 180,E1 -13790.863,E2 -13790.863} C_VEL
LIN {X 0,Y 346.595,Z 221.959,A -85,B 0,C 180,E1 -13790.94,E2 -13790.94} C_VEL
LIN {X 0,Y 346.876,Z 217.617,A -85,B 0,C 180,E1 -13794.252,E2 -13794.252} C_VEL
LIN {X 0,Y 347.218,Z 213.13,A -85,B 0,C 180,E1 -13797.745,E2 -13797.745} C_VEL
LIN {X 0,Y 347.718,Z 208.221,A -85,B 0,C 180,E1 -13801.702,E2 -13801.702} C_VEL
LIN {X 0,Y 348.288,Z 203.388,A -85,B 0,C 180,E1 -13805.815,E2 -13805.815} C_VEL
LIN {X 0,Y 348.694,Z 200.205,A -85,B 0,C 180,E1 -13808.668,E2 -13808.668} C_VEL
LIN {X 0,Y 348.99,Z 197.085,A -85,B 0,C 180,E1 -13811.648,E2 -13811.648} C_VEL
LIN {X 0,Y 348.815,Z 193.999,A -85,B 0,C 180,E1 -13814.844,E2 -13814.844} C_VEL
LIN {X 0,Y 348.393,Z 190.987,A -85,B 0,C 180,E1 -13818.277,E2 -13818.277} C_VEL
LIN {X 0,Y 348.04,Z 188.613,A -85,B 0,C 180,E1 -13821.245,E2 -13821.245} C_VEL
LIN {X 0,Y 347.786,Z 186.666,A -85,B 0,C 180,E1 -13824.124,E2 -13824.124} C_VEL
LIN {X 0,Y 347.737,Z 186.668,A -85,B 0,C 180,E1 -13828.085,E2 -13828.085} C_VEL
LIN {X 0,Y 347.776,Z 186.664,A -85,B 0,C 180,E1 -13830.987,E2 -13830.987} C_VEL
LIN {X 0,Y 347.828,Z 186.655,A -85,B 0,C 180,E1 -13833.607,E2 -13833.607} C_VEL
LIN {X 0,Y 347.786,Z 186.664,A -85,B 0,C 180,E1 -13836.161,E2 -13836.161} C_VEL
LIN {X 0,Y 347.809,Z 186.66,A -85,B 0,C 180,E1 -13839.909,E2 -13839.909} C_VEL
LIN {X 0,Y 347.863,Z 186.655,A -85,B 0,C 180,E1 -13842.358,E2 -13842.358} C_VEL
LIN {X 0,Y 347.894,Z 186.651,A -85,B 0,C 180,E1 -13845.97,E2 -13845.97} C_VEL
LIN {X 0,Y 347.924,Z 186.645,A -85,B 0,C 180,E1 -13849.525,E2 -13849.525} C_VEL
LIN {X 0,Y 348.086,Z 186.623,A -85,B 0,C 180,E1 -13853.041,E2 -13853.041} C_VEL
LIN {X 0,Y 348.2,Z 186.614,A -85,B 0,C 180,E1 -13857.686,E2 -13857.686} C_VEL
LIN {X 0,Y 348.341,Z 186.593,A -85,B 0,C 180,E1 -13859.999,E2 -13859.999} C_VEL
LIN {X 0,Y 348.201,Z 186.607,A -85,B 0,C 180,E1 -13862.313,E2 -13862.313} C_VEL
LIN {X 0,Y 348.087,Z 186.624,A -85,B 0,C 180,E1 -13866.957,E2 -13866.957} C_VEL
LIN {X 0,Y 347.923,Z 186.643,A -85,B 0,C 180,E1 -13870.474,E2 -13870.474} C_VEL
LIN {X 0,Y 347.893,Z 186.647,A -85,B 0,C 180,E1 -13874.149,E2 -13874.149} C_VEL
LIN {X 0,Y 347.885,Z 186.648,A -85,B 0,C 180,E1 -13878.29,E2 -13878.29} C_VEL
LIN {X 0,Y 347.783,Z 186.661,A -85,B 0,C 180,E1 -13881.635,E2 -13881.635} C_VEL
LIN {X 0,Y 347.807,Z 186.662,A -85,B 0,C 180,E1 -13885.108,E2 -13885.108} C_VEL
LIN {X 0,Y 347.806,Z 186.658,A -85,B 0,C 180,E1 -13887.693,E2 -13887.693} C_VEL
LIN {X 0,Y 347.759,Z 186.666,A -85,B 0,C 180,E1 -13890.346,E2 -13890.346} C_VEL
LIN {X 0,Y 347.739,Z 186.67,A -85,B 0,C 180,E1 -13894.464,E2 -13894.464} C_VEL
LIN {X 0,Y 347.771,Z 186.663,A -85,B 0,C 180,E1 -13897.989,E2 -13897.989} C_VEL
LIN {X 0,Y 347.761,Z 186.664,A -85,B 0,C 180,E1 -13901.828,E2 -13901.828} C_VEL
LIN {X 0,Y 347.702,Z 186.671,A -85,B 0,C 180,E1 -13905.026,E2 -13905.026} C_VEL
LIN {X 0,Y 347.745,Z 186.67,A -85,B 0,C 180,E1 -13908.397,E2 -13908.397} C_VEL
LIN {X 0,Y 347.769,Z 186.667,A -85,B 0,C 180,E1 -13912.011,E2 -13912.011} C_VEL
LIN {X 0,Y 347.74,Z 186.668,A -85,B 0,C 180,E1 -13915.536,E2 -13915.536} C_VEL
LIN {X 0,Y 347.759,Z 186.666,A -85,B 0,C 180,E1 -13918.302,E2 -13918.302} C_VEL
LIN {X 0,Y 347.801,Z 186.658,A -85,B 0,C 180,E1 -13920.99,E2 -13920.99} C_VEL
LIN {X 0,Y 347.828,Z 186.659,A -85,B 0,C 180,E1 -13923.608,E2 -13923.608} C_VEL
LIN {X 0,Y 347.784,Z 186.663,A -85,B 0,C 180,E1 -13926.162,E2 -13926.162} C_VEL
LIN {X 0,Y 347.814,Z 186.661,A -85,B 0,C 180,E1 -13929.91,E2 -13929.91} C_VEL
LIN {X 0,Y 347.84,Z 186.657,A -85,B 0,C 180,E1 -13931.024,E2 -13931.024} C_VEL
LIN {X 0,Y 348.761,Z 189.365,A -85,B 0,C 180,E1 -13931.28,E2 -13931.28} C_VEL
LIN {X 0,Y 350.961,Z 191.677,A -85,B 0,C 180,E1 -13931.757,E2 -13931.757} C_VEL
LIN {X 0,Y 351.651,Z 192.522,A -85,B 0,C 180,E1 -13931.915,E2 -13931.915} C_VEL
LIN {X 0,Y 353.957,Z 195.838,A -85,B 0,C 180,E1 -13932.456,E2 -13932.456} C_VEL
LIN {X 0,Y 356.184,Z 198.068,A -85,B 0,C 180,E1 -13932.985,E2 -13932.985} C_VEL
LIN {X 0,Y 358.881,Z 201.48,A -85,B 0,C 180,E1 -13933.649,E2 -13933.649} C_VEL
LIN {X 0,Y 361.214,Z 203.691,A -85,B 0,C 180,E1 -13934.252,E2 -13934.252} C_VEL
LIN {X 0,Y 364.424,Z 207.405,A -85,B 0,C 180,E1 -13935.115,E2 -13935.115} C_VEL
LIN {X 0,Y 367.188,Z 209.737,A -85,B 0,C 180,E1 -13935.883,E2 -13935.883} C_VEL
LIN {X 0,Y 370.231,Z 213.265,A -85,B 0,C 180,E1 -13936.833,E2 -13936.833} C_VEL
LIN {X 0,Y 374.052,Z 216.349,A -85,B 0,C 180,E1 -13938.073,E2 -13938.073} C_VEL
LIN {X 0,Y 376.845,Z 219.443,A -85,B 0,C 180,E1 -13939.116,E2 -13939.116} C_VEL
LIN {X 0,Y 380.1,Z 221.907,A -85,B 0,C 180,E1 -13940.421,E2 -13940.421} C_VEL
LIN {X 0,Y 381.94,Z 223.03,A -85,B 0,C 180,E1 -13941.235,E2 -13941.235} C_VEL
LIN {X 0,Y 384.566,Z 226.122,A -85,B 0,C 180,E1 -13942.65,E2 -13942.65} C_VEL
LIN {X 0,Y 386.682,Z 227.954,A -85,B 0,C 180,E1 -13944.001,E2 -13944.001} C_VEL
LIN {X 0,Y 388.71,Z 229.139,A -85,B 0,C 180,E1 -13945.593,E2 -13945.593} C_VEL
LIN {X 0,Y 389.939,Z 229.474,A -85,B 0,C 180,E1 -13946.901,E2 -13946.901} C_VEL
LIN {X 0,Y 390.625,Z 229.63,A -85,B 0,C 180,E1 -13947.938,E2 -13947.938} C_VEL
LIN {X 0,Y 391.046,Z 229.675,A -85,B 0,C 180,E1 -13948.97,E2 -13948.97} C_VEL
LIN {X 0,Y 391.184,Z 229.718,A -85,B 0,C 180,E1 -13950,E2 -13950} C_VEL
LIN {X 0,Y 391.048,Z 229.661,A -85,B 0,C 180,E1 -13951.03,E2 -13951.03} C_VEL
LIN {X 0,Y 390.625,Z 229.62,A -85,B 0,C 180,E1 -13952.062,E2 -13952.062} C_VEL
LIN {X 0,Y 389.525,Z 229.371,A -85,B 0,C 180,E1 -13953.61,E2 -13953.61} C_VEL
LIN {X 0,Y 387.765,Z 228.68,A -85,B 0,C 180,E1 -13955.199,E2 -13955.199} C_VEL
LIN {X 0,Y 385.352,Z 226.883,A -85,B 0,C 180,E1 -13956.867,E2 -13956.867} C_VEL
LIN {X 0,Y 382.721,Z 224.046,A -85,B 0,C 180,E1 -13958.361,E2 -13958.361} C_VEL
LIN {X 0,Y 381.492,Z 222.586,A -85,B 0,C 180,E1 -13958.983,E2 -13958.983} C_VEL
LIN {X 0,Y 378.356,Z 220.726,A -85,B 0,C 180,E1 -13960.292,E2 -13960.292} C_VEL
LIN {X 0,Y 375.221,Z 217.793,A -85,B 0,C 180,E1 -13961.498,E2 -13961.498} C_VEL
LIN {X 0,Y 373.073,Z 215.444,A -85,B 0,C 180,E1 -13962.267,E2 -13962.267} C_VEL
LIN {X 0,Y 369.723,Z 212.779,A -85,B 0,C 180,E1 -13963.326,E2 -13963.326} C_VEL
LIN {X 0,Y 366.192,Z 208.784,A -85,B 0,C 180,E1 -13964.4,E2 -13964.4} C_VEL
LIN {X 0,Y 362.953,Z 205.908,A -85,B 0,C 180,E1 -13965.279,E2 -13965.279} C_VEL
LIN {X 0,Y 360.503,Z 202.837,A -85,B 0,C 180,E1 -13965.94,E2 -13965.94} C_VEL
LIN {X 0,Y 357.57,Z 200.079,A -85,B 0,C 180,E1 -13966.664,E2 -13966.664} C_VEL
LIN {X 0,Y 355.394,Z 197.109,A -85,B 0,C 180,E1 -13967.209,E2 -13967.209} C_VEL
LIN {X 0,Y 352.738,Z 194.374,A -85,B 0,C 180,E1 -13967.823,E2 -13967.823} C_VEL
LIN {X 0,Y 351.102,Z 191.767,A -85,B 0,C 180,E1 -13968.213,E2 -13968.213} C_VEL
LIN {X 0,Y 348.922,Z 189.629,A -85,B 0,C 180,E1 -13968.682,E2 -13968.682} C_VEL
LIN {X 0,Y 347.945,Z 187.339,A -85,B 0,C 180,E1 -13968.931,E2 -13968.931} C_VEL
LIN {X 0,Y 347.829,Z 186.66,A -85,B 0,C 180,E1 -13969.014,E2 -13969.014} C_VEL
LIN {X 0,Y 347.77,Z 186.666,A -85,B 0,C 180,E1 -13972.579,E2 -13972.579} C_VEL
LIN {X 0,Y 347.808,Z 186.658,A -85,B 0,C 180,E1 -13975.108,E2 -13975.108} C_VEL
LIN {X 0,Y 347.808,Z 186.659,A -85,B 0,C 180,E1 -13977.694,E2 -13977.694} C_VEL
LIN {X 0,Y 347.766,Z 186.666,A -85,B 0,C 180,E1 -13980.346,E2 -13980.346} C_VEL
LIN {X 0,Y 347.743,Z 186.671,A -85,B 0,C 180,E1 -13984.044,E2 -13984.044} C_VEL
LIN {X 0,Y 347.761,Z 186.664,A -85,B 0,C 180,E1 -13987.32,E2 -13987.32} C_VEL
LIN {X 0,Y 347.75,Z 186.666,A -85,B 0,C 180,E1 -13990.294,E2 -13990.294} C_VEL
LIN {X 0,Y 347.738,Z 186.669,A -85,B 0,C 180,E1 -13993.405,E2 -13993.405} C_VEL
LIN {X 0,Y 347.726,Z 186.668,A -85,B 0,C 180,E1 -13996.685,E2 -13996.685} C_VEL
LIN {X 0,Y 347.752,Z 186.665,A -85,B 0,C 180,E1 -14000.171,E2 -14000.171} C_VEL
LIN {X 0,Y 347.765,Z 186.664,A -85,B 0,C 180,E1 -14003.935,E2 -14003.935} C_VEL
LIN {X 0,Y 347.727,Z 186.67,A -85,B 0,C 180,E1 -14006.928,E2 -14006.928} C_VEL
LIN {X 0,Y 347.75,Z 186.666,A -85,B 0,C 180,E1 -14009.548,E2 -14009.548} C_VEL
LIN {X 0,Y 347.143,Z 186.747,A -85,B 0,C 180,E1 -14010.516,E2 -14010.516} C_VEL
LIN {X 0,Y 344.32,Z 187.097,A -85,B 0,C 180,E1 -14012.091,E2 -14012.091} C_VEL
LIN {X 0,Y 341.891,Z 187.398,A -85,B 0,C 180,E1 -14013.365,E2 -14013.365} C_VEL
LIN {X 0,Y 340.842,Z 187.525,A -85,B 0,C 180,E1 -14014.352,E2 -14014.352} C_VEL
LIN {X 0,Y 340.756,Z 187.537,A -85,B 0,C 180,E1 -14014.686,E2 -14014.686} C_VEL
LIN {X 0,Y 340.736,Z 187.539,A -85,B 0,C 180,E1 -14018.207,E2 -14018.207} C_VEL
LIN {X 0,Y 340.852,Z 187.524,A -85,B 0,C 180,E1 -14021.985,E2 -14021.985} C_VEL
LIN {X 0,Y 340.864,Z 187.522,A -85,B 0,C 180,E1 -14025.706,E2 -14025.706} C_VEL
LIN {X 0,Y 340.865,Z 187.522,A -85,B 0,C 180,E1 -14029.307,E2 -14029.307} C_VEL
LIN {X 0,Y 341.054,Z 187.501,A -85,B 0,C 180,E1 -14032.898,E2 -14032.898} C_VEL
LIN {X 0,Y 341.163,Z 187.483,A -85,B 0,C 180,E1 -14037.639,E2 -14037.639} C_VEL
LIN {X 0,Y 341.291,Z 187.47,A -85,B 0,C 180,E1 -14040.001,E2 -14040.001} C_VEL
LIN {X 0,Y 341.162,Z 187.49,A -85,B 0,C 180,E1 -14042.362,E2 -14042.362} C_VEL
LIN {X 0,Y 341.054,Z 187.499,A -85,B 0,C 180,E1 -14047.103,E2 -14047.103} C_VEL
LIN {X 0,Y 340.867,Z 187.523,A -85,B 0,C 180,E1 -14050.695,E2 -14050.695} C_VEL
LIN {X 0,Y 340.86,Z 187.525,A -85,B 0,C 180,E1 -14054.326,E2 -14054.326} C_VEL
LIN {X 0,Y 340.834,Z 187.527,A -85,B 0,C 180,E1 -14058.467,E2 -14058.467} C_VEL
LIN {X 0,Y 340.751,Z 187.541,A -85,B 0,C 180,E1 -14061.858,E2 -14061.858} C_VEL
LIN {X 0,Y 340.77,Z 187.539,A -85,B 0,C 180,E1 -14065.665,E2 -14065.665} C_VEL
LIN {X 0,Y 340.726,Z 187.54,A -85,B 0,C 180,E1 -14068.322,E2 -14068.322} C_VEL
LIN {X 0,Y 340.696,Z 187.547,A -85,B 0,C 180,E1 -14071.046,E2 -14071.046} C_VEL
LIN {X 0,Y 340.716,Z 187.546,A -85,B 0,C 180,E1 -14075.28,E2 -14075.28} C_VEL
LIN {X 0,Y 340.817,Z 188.245,A -85,B 0,C 180,E1 -14076.728,E2 -14076.728} C_VEL
LIN {X 0,Y 341.24,Z 190.968,A -85,B 0,C 180,E1 -14080.357,E2 -14080.357} C_VEL
LIN {X 0,Y 341.638,Z 193.976,A -85,B 0,C 180,E1 -14083.946,E2 -14083.946} C_VEL
LIN {X 0,Y 341.925,Z 197.033,A -85,B 0,C 180,E1 -14087.291,E2 -14087.291} C_VEL
LIN {X 0,Y 341.777,Z 200.141,A -85,B 0,C 180,E1 -14090.398,E2 -14090.398} C_VEL
LIN {X 0,Y 341.337,Z 203.379,A -85,B 0,C 180,E1 -14093.418,E2 -14093.418} C_VEL
LIN {X 0,Y 340.907,Z 206.487,A -85,B 0,C 180,E1 -14096.178,E2 -14096.178} C_VEL
LIN {X 0,Y 340.392,Z 211.143,A -85,B 0,C 180,E1 -14100.132,E2 -14100.132} C_VEL
LIN {X 0,Y 340.068,Z 214.622,A -85,B 0,C 180,E1 -14102.957,E2 -14102.957} C_VEL
LIN {X 0,Y 339.648,Z 219.553,A -85,B 0,C 180,E1 -14106.85,E2 -14106.85} C_VEL
LIN {X 0,Y 339.524,Z 221.796,A -85,B 0,C 180,E1 -14108.627,E2 -14108.627} C_VEL
LIN {X 0,Y 341.965,Z 232.723,A -85,B 0,C 180,E1 -14109.202,E2 -14109.202} C_VEL
LIN {X 0,Y 343.929,Z 243.148,A -85,B 0,C 180,E1 -14109.885,E2 -14109.885} C_VEL
LIN {X 0,Y 345.392,Z 253.943,A -85,B 0,C 180,E1 -14110.735,E2 -14110.735} C_VEL
LIN {X 0,Y 346.092,Z 260.54,A -85,B 0,C 180,E1 -14111.348,E2 -14111.348} C_VEL
LIN {X 0,Y 345.18,Z 269.539,A -85,B 0,C 180,E1 -14112.218,E2 -14112.218} C_VEL
LIN {X 0,Y 344.189,Z 278.27,A -85,B 0,C 180,E1 -14113.237,E2 -14113.237} C_VEL
LIN {X 0,Y 343.272,Z 286.46,A -85,B 0,C 180,E1 -14114.386,E2 -14114.386} C_VEL
LIN {X 0,Y 342.285,Z 294.52,A -85,B 0,C 180,E1 -14115.736,E2 -14115.736} C_VEL
LIN {X 0,Y 341.507,Z 300.472,A -85,B 0,C 180,E1 -14116.917,E2 -14116.917} C_VEL
LIN {X 0,Y 340.684,Z 306.791,A -85,B 0,C 180,E1 -14118.397,E2 -14118.397} C_VEL
LIN {X 0,Y 340.105,Z 312.057,A -85,B 0,C 180,E1 -14119.884,E2 -14119.884} C_VEL
LIN {X 0,Y 339.57,Z 317.19,A -85,B 0,C 180,E1 -14121.67,E2 -14121.67} C_VEL
LIN {X 0,Y 339.251,Z 321.181,A -85,B 0,C 180,E1 -14123.458,E2 -14123.458} C_VEL
LIN {X 0,Y 339.116,Z 324.133,A -85,B 0,C 180,E1 -14125.245,E2 -14125.245} C_VEL
LIN {X 0,Y 338.999,Z 326.58,A -85,B 0,C 180,E1 -14127.624,E2 -14127.624} C_VEL
LIN {X 0,Y 338.999,Z 327.169,A -85,B 0,C 180,E1 -14128.812,E2 -14128.812} C_VEL
LIN {X 0,Y 338.999,Z 327.169,A -85,B 0,C 180,E1 -14131.188,E2 -14131.188} C_VEL
LIN {X 0,Y 338.999,Z 326.58,A -85,B 0,C 180,E1 -14132.376,E2 -14132.376} C_VEL
LIN {X 0,Y 339.116,Z 324.133,A -85,B 0,C 180,E1 -14134.755,E2 -14134.755} C_VEL
LIN {X 0,Y 339.261,Z 321.181,A -85,B 0,C 180,E1 -14136.542,E2 -14136.542} C_VEL
LIN {X 0,Y 339.57,Z 317.19,A -85,B 0,C 180,E1 -14138.33,E2 -14138.33} C_VEL
LIN {X 0,Y 340.105,Z 312.057,A -85,B 0,C 180,E1 -14140.116,E2 -14140.116} C_VEL
LIN {X 0,Y 340.683,Z 306.791,A -85,B 0,C 180,E1 -14141.603,E2 -14141.603} C_VEL
LIN {X 0,Y 341.506,Z 300.472,A -85,B 0,C 180,E1 -14143.083,E2 -14143.083} C_VEL
LIN {X 0,Y 342.277,Z 294.519,A -85,B 0,C 180,E1 -14144.264,E2 -14144.264} C_VEL
LIN {X 0,Y 343.302,Z 286.338,A -85,B 0,C 180,E1 -14145.632,E2 -14145.632} C_VEL
LIN {X 0,Y 344.151,Z 278.269,A -85,B 0,C 180,E1 -14146.765,E2 -14146.765} C_VEL
LIN {X 0,Y 345.209,Z 269.54,A -85,B 0,C 180,E1 -14147.781,E2 -14147.781} C_VEL
LIN {X 0,Y 346.084,Z 260.54,A -85,B 0,C 180,E1 -14148.653,E2 -14148.653} C_VEL
LIN {X 0,Y 344.989,Z 250.46,A -85,B 0,C 180,E1 -14149.554,E2 -14149.554} C_VEL
LIN {X 0,Y 343.611,Z 241.219,A -85,B 0,C 180,E1 -14150.25,E2 -14150.25} C_VEL
LIN {X 0,Y 341.513,Z 230.552,A -85,B 0,C 180,E1 -14150.924,E2 -14150.924} C_VEL
LIN {X 0,Y 339.53,Z 221.771,A -85,B 0,C 180,E1 -14151.393,E2 -14151.393} C_VEL
LIN {X 0,Y 339.811,Z 217.829,A -85,B 0,C 180,E1 -14154.492,E2 -14154.492} C_VEL
LIN {X 0,Y 340.214,Z 212.994,A -85,B 0,C 180,E1 -14158.367,E2 -14158.367} C_VEL
LIN {X 0,Y 340.721,Z 208.095,A -85,B 0,C 180,E1 -14162.431,E2 -14162.431} C_VEL
LIN {X 0,Y 341.135,Z 204.877,A -85,B 0,C 180,E1 -14165.229,E2 -14165.229} C_VEL
LIN {X 0,Y 341.639,Z 201.211,A -85,B 0,C 180,E1 -14168.581,E2 -14168.581} C_VEL
LIN {X 0,Y 341.913,Z 198.575,A -85,B 0,C 180,E1 -14171.128,E2 -14171.128} C_VEL
LIN {X 0,Y 341.824,Z 195.488,A -85,B 0,C 180,E1 -14174.35,E2 -14174.35} C_VEL
LIN {X 0,Y 341.409,Z 192.457,A -85,B 0,C 180,E1 -14177.822,E2 -14177.822} C_VEL
LIN {X 0,Y 341.155,Z 190.454,A -85,B 0,C 180,E1 -14180.31,E2 -14180.31} C_VEL
LIN {X 0,Y 340.791,Z 188.055,A -85,B 0,C 180,E1 -14183.54,E2 -14183.54} C_VEL
LIN {X 0,Y 340.716,Z 187.548,A -85,B 0,C 180,E1 -14184.72,E2 -14184.72} C_VEL
LIN {X 0,Y 340.696,Z 187.547,A -85,B 0,C 180,E1 -14188.954,E2 -14188.954} C_VEL
LIN {X 0,Y 340.801,Z 187.532,A -85,B 0,C 180,E1 -14193.019,E2 -14193.019} C_VEL
LIN {X 0,Y 340.753,Z 187.537,A -85,B 0,C 180,E1 -14195.638,E2 -14195.638} C_VEL
LIN {X 0,Y 340.742,Z 187.538,A -85,B 0,C 180,E1 -14199.473,E2 -14199.473} C_VEL
LIN {X 0,Y 340.854,Z 187.527,A -85,B 0,C 180,E1 -14201.983,E2 -14201.983} C_VEL
LIN {X 0,Y 340.866,Z 187.524,A -85,B 0,C 180,E1 -14205.704,E2 -14205.704} C_VEL
LIN {X 0,Y 340.867,Z 187.523,A -85,B 0,C 180,E1 -14209.305,E2 -14209.305} C_VEL
LIN {X 0,Y 341.054,Z 187.499,A -85,B 0,C 180,E1 -14212.897,E2 -14212.897} C_VEL
LIN {X 0,Y 341.162,Z 187.49,A -85,B 0,C 180,E1 -14217.638,E2 -14217.638} C_VEL
LIN {X 0,Y 341.291,Z 187.47,A -85,B 0,C 180,E1 -14219.999,E2 -14219.999} C_VEL
LIN {X 0,Y 341.163,Z 187.483,A -85,B 0,C 180,E1 -14222.361,E2 -14222.361} C_VEL
LIN {X 0,Y 341.054,Z 187.501,A -85,B 0,C 180,E1 -14227.102,E2 -14227.102} C_VEL
LIN {X 0,Y 340.865,Z 187.522,A -85,B 0,C 180,E1 -14230.693,E2 -14230.693} C_VEL
LIN {X 0,Y 340.858,Z 187.523,A -85,B 0,C 180,E1 -14234.324,E2 -14234.324} C_VEL
LIN {X 0,Y 340.831,Z 187.527,A -85,B 0,C 180,E1 -14238.466,E2 -14238.466} C_VEL
LIN {X 0,Y 340.748,Z 187.537,A -85,B 0,C 180,E1 -14241.857,E2 -14241.857} C_VEL
LIN {X 0,Y 340.767,Z 187.535,A -85,B 0,C 180,E1 -14245.664,E2 -14245.664} C_VEL
LIN {X 0,Y 340.737,Z 187.54,A -85,B 0,C 180,E1 -14248.319,E2 -14248.319} C_VEL
LIN {X 0,Y 340.698,Z 187.546,A -85,B 0,C 180,E1 -14251.044,E2 -14251.044} C_VEL
LIN {X 0,Y 340.713,Z 187.542,A -85,B 0,C 180,E1 -14255.279,E2 -14255.279} C_VEL
LIN {X 0,Y 340.712,Z 187.546,A -85,B 0,C 180,E1 -14258.388,E2 -14258.388} C_VEL
LIN {X 0,Y 340.724,Z 187.542,A -85,B 0,C 180,E1 -14262.051,E2 -14262.051} C_VEL
LIN {X 0,Y 340.647,Z 187.555,A -85,B 0,C 180,E1 -14266.227,E2 -14266.227} C_VEL
LIN {X 0,Y 340.683,Z 187.547,A -85,B 0,C 180,E1 -14269.753,E2 -14269.753} C_VEL
LIN {X 0,Y 340.7,Z 187.543,A -85,B 0,C 180,E1 -14273.259,E2 -14273.259} C_VEL
LIN {X 0,Y 340.69,Z 187.549,A -85,B 0,C 180,E1 -14276.154,E2 -14276.154} C_VEL
LIN {X 0,Y 340.771,Z 187.536,A -85,B 0,C 180,E1 -14280.333,E2 -14280.333} C_VEL
LIN {X 0,Y 340.801,Z 187.531,A -85,B 0,C 180,E1 -14283.02,E2 -14283.02} C_VEL
LIN {X 0,Y 340.725,Z 187.541,A -85,B 0,C 180,E1 -14286.927,E2 -14286.927} C_VEL
LIN {X 0,Y 340.77,Z 187.539,A -85,B 0,C 180,E1 -14289.83,E2 -14289.83} C_VEL
LIN {X 0,Y 341.841,Z 190.504,A -85,B 0,C 180,E1 -14290.115,E2 -14290.115} C_VEL
LIN {X 0,Y 344.235,Z 193.109,A -85,B 0,C 180,E1 -14290.593,E2 -14290.593} C_VEL
LIN {X 0,Y 346.385,Z 196.299,A -85,B 0,C 180,E1 -14291.057,E2 -14291.057} C_VEL
LIN {X 0,Y 348.434,Z 198.477,A -85,B 0,C 180,E1 -14291.494,E2 -14291.494} C_VEL
LIN {X 0,Y 351.083,Z 201.947,A -85,B 0,C 180,E1 -14292.099,E2 -14292.099} C_VEL
LIN {X 0,Y 353.191,Z 204.033,A -85,B 0,C 180,E1 -14292.561,E2 -14292.561} C_VEL
LIN {X 0,Y 356.4,Z 207.856,A -85,B 0,C 180,E1 -14293.346,E2 -14293.346} C_VEL
LIN {X 0,Y 358.92,Z 210.288,A -85,B 0,C 180,E1 -14293.953,E2 -14293.953} C_VEL
LIN {X 0,Y 362.355,Z 214.03,A -85,B 0,C 180,E1 -14294.862,E2 -14294.862} C_VEL
LIN {X 0,Y 365.004,Z 216.311,A -85,B 0,C 180,E1 -14295.576,E2 -14295.576} C_VEL
LIN {X 0,Y 368.716,Z 220.25,A -85,B 0,C 180,E1 -14296.684,E2 -14296.684} C_VEL
LIN {X 0,Y 372.223,Z 223.043,A -85,B 0,C 180,E1 -14297.793,E2 -14297.793} C_VEL
LIN {X 0,Y 375.555,Z 226.51,A -85,B 0,C 180,E1 -14299.01,E2 -14299.01} C_VEL
LIN {X 0,Y 379.049,Z 228.975,A -85,B 0,C 180,E1 -14300.394,E2 -14300.394} C_VEL
LIN {X 0,Y 380.499,Z 229.865,A -85,B 0,C 180,E1 -14301.028,E2 -14301.028} C_VEL
LIN {X 0,Y 383.023,Z 232.827,A -85,B 0,C 180,E1 -14302.389,E2 -14302.389} C_VEL
LIN {X 0,Y 385.458,Z 234.922,A -85,B 0,C 180,E1 -14303.917,E2 -14303.917} C_VEL
LIN {X 0,Y 387.661,Z 236.156,A -85,B 0,C 180,E1 -14305.633,E2 -14305.633} C_VEL
LIN {X 0,Y 388.858,Z 236.483,A -85,B 0,C 180,E1 -14306.892,E2 -14306.892} C_VEL
LIN {X 0,Y 389.963,Z 236.691,A -85,B 0,C 180,E1 -14308.967,E2 -14308.967} C_VEL
LIN {X 0,Y 390.106,Z 236.735,A -85,B 0,C 180,E1 -14310,E2 -14310} C_VEL
LIN {X 0,Y 389.963,Z 236.673,A -85,B 0,C 180,E1 -14311.033,E2 -14311.033} C_VEL
LIN {X 0,Y 389.54,Z 236.636,A -85,B 0,C 180,E1 -14312.068,E2 -14312.068} C_VEL
LIN {X 0,Y 388.416,Z 236.367,A -85,B 0,C 180,E1 -14313.62,E2 -14313.62} C_VEL
LIN {X 0,Y 386.651,Z 235.705,A -85,B 0,C 180,E1 -14315.214,E2 -14315.214} C_VEL
LIN {X 0,Y 384.088,Z 233.833,A -85,B 0,C 180,E1 -14316.986,E2 -14316.986} C_VEL
LIN {X 0,Y 381.314,Z 230.901,A -85,B 0,C 180,E1 -14318.546,E2 -14318.546} C_VEL
LIN {X 0,Y 380.063,Z 229.448,A -85,B 0,C 180,E1 -14319.168,E2 -14319.168} C_VEL
LIN {X 0,Y 376.824,Z 227.48,A -85,B 0,C 180,E1 -14320.511,E2 -14320.511} C_VEL
LIN {X 0,Y 373.455,Z 224.473,A -85,B 0,C 180,E1 -14321.767,E2 -14321.767} C_VEL
LIN {X 0,Y 371.175,Z 222.06,A -85,B 0,C 180,E1 -14322.554,E2 -14322.554} C_VEL
LIN {X 0,Y 367.554,Z 219.155,A -85,B 0,C 180,E1 -14323.67,E2 -14323.67} C_VEL
LIN {X 0,Y 363.729,Z 215.052,A -85,B 0,C 180,E1 -14324.784,E2 -14324.784} C_VEL
LIN {X 0,Y 360.231,Z 211.902,A -85,B 0,C 180,E1 -14325.69,E2 -14325.69} C_VEL
LIN {X 0,Y 357.641,Z 208.882,A -85,B 0,C 180,E1 -14326.368,E2 -14326.368} C_VEL
LIN {X 0,Y 354.27,Z 205.535,A -85,B 0,C 180,E1 -14327.171,E2 -14327.171} C_VEL
LIN {X 0,Y 352.212,Z 202.967,A -85,B 0,C 180,E1 -14327.658,E2 -14327.658} C_VEL
LIN {X 0,Y 349.106,Z 199.555,A -85,B 0,C 180,E1 -14328.349,E2 -14328.349} C_VEL
LIN {X 0,Y 347.585,Z 197.443,A -85,B 0,C 180,E1 -14328.694,E2 -14328.694} C_VEL
LIN {X 0,Y 345.115,Z 194.681,A -85,B 0,C 180,E1 -14329.211,E2 -14329.211} C_VEL
LIN {X 0,Y 343.719,Z 192.459,A -85,B 0,C 180,E1 -14329.512,E2 -14329.512} C_VEL
LIN {X 0,Y 341.671,Z 190.212,A -85,B 0,C 180,E1 -14329.921,E2 -14329.921} C_VEL
LIN {X 0,Y 340.773,Z 187.539,A -85,B 0,C 180,E1 -14330.188,E2 -14330.188} C_VEL
LIN {X 0,Y 340.725,Z 187.541,A -85,B 0,C 180,E1 -14333.073,E2 -14333.073} C_VEL
LIN {X 0,Y 340.801,Z 187.531,A -85,B 0,C 180,E1 -14336.98,E2 -14336.98} C_VEL
LIN {X 0,Y 340.761,Z 187.54,A -85,B 0,C 180,E1 -14339.979,E2 -14339.979} C_VEL
LIN {X 0,Y 340.69,Z 187.549,A -85,B 0,C 180,E1 -14343.846,E2 -14343.846} C_VEL
LIN {X 0,Y 340.702,Z 187.543,A -85,B 0,C 180,E1 -14346.741,E2 -14346.741} C_VEL
LIN {X 0,Y 340.704,Z 187.544,A -85,B 0,C 180,E1 -14350.251,E2 -14350.251} C_VEL
LIN {X 0,Y 340.706,Z 187.542,A -85,B 0,C 180,E1 -14352.899,E2 -14352.899} C_VEL
LIN {X 0,Y 340.696,Z 187.545,A -85,B 0,C 180,E1 -14357.1,E2 -14357.1} C_VEL
LIN {X 0,Y 340.704,Z 187.543,A -85,B 0,C 180,E1 -14360.249,E2 -14360.249} C_VEL
LIN {X 0,Y 340.705,Z 187.546,A -85,B 0,C 180,E1 -14363.559,E2 -14363.559} C_VEL
LIN {X 0,Y 340.686,Z 187.545,A -85,B 0,C 180,E1 -14366.154,E2 -14366.154} C_VEL
LIN {X 0,Y 340.769,Z 187.534,A -85,B 0,C 180,E1 -14370.333,E2 -14370.333} C_VEL
LIN {X 0,Y 340.799,Z 187.535,A -85,B 0,C 180,E1 -14373.02,E2 -14373.02} C_VEL
LIN {X 0,Y 340.756,Z 187.537,A -85,B 0,C 180,E1 -14374.686,E2 -14374.686} C_VEL
LIN {X 0,Y 340.074,Z 187.625,A -85,B 0,C 180,E1 -14375.673,E2 -14375.673} C_VEL
LIN {X 0,Y 337.181,Z 187.985,A -85,B 0,C 180,E1 -14377.278,E2 -14377.278} C_VEL
LIN {X 0,Y 334.761,Z 188.285,A -85,B 0,C 180,E1 -14378.578,E2 -14378.578} C_VEL
LIN {X 0,Y 333.76,Z 188.407,A -85,B 0,C 180,E1 -14379.584,E2 -14379.584} C_VEL
LIN {X 0,Y 333.699,Z 188.414,A -85,B 0,C 180,E1 -14379.925,E2 -14379.925} C_VEL
LIN {X 0,Y 333.741,Z 188.415,A -85,B 0,C 180,E1 -14382.854,E2 -14382.854} C_VEL
LIN {X 0,Y 333.791,Z 188.408,A -85,B 0,C 180,E1 -14386.609,E2 -14386.609} C_VEL
LIN {X 0,Y 333.845,Z 188.399,A -85,B 0,C 180,E1 -14390.305,E2 -14390.305} C_VEL
LIN {X 0,Y 334.001,Z 188.381,A -85,B 0,C 180,E1 -14392.748,E2 -14392.748} C_VEL
LIN {X 0,Y 333.803,Z 188.401,A -85,B 0,C 180,E1 -14395.17,E2 -14395.17} C_VEL
LIN {X 0,Y 334.1,Z 188.361,A -85,B 0,C 180,E1 -14397.589,E2 -14397.589} C_VEL
LIN {X 0,Y 334.242,Z 188.348,A -85,B 0,C 180,E1 -14400.001,E2 -14400.001} C_VEL
LIN {X 0,Y 334.1,Z 188.369,A -85,B 0,C 180,E1 -14402.412,E2 -14402.412} C_VEL
LIN {X 0,Y 334.009,Z 188.381,A -85,B 0,C 180,E1 -14406.04,E2 -14406.04} C_VEL
LIN {X 0,Y 333.955,Z 188.385,A -85,B 0,C 180,E1 -14408.472,E2 -14408.472} C_VEL
LIN {X 0,Y 333.787,Z 188.408,A -85,B 0,C 180,E1 -14412.155,E2 -14412.155} C_VEL
LIN {X 0,Y 333.774,Z 188.411,A -85,B 0,C 180,E1 -14415.887,E2 -14415.887} C_VEL
LIN {X 0,Y 333.793,Z 188.404,A -85,B 0,C 180,E1 -14418.656,E2 -14418.656} C_VEL
LIN {X 0,Y 333.69,Z 188.417,A -85,B 0,C 180,E1 -14422.279,E2 -14422.279} C_VEL
LIN {X 0,Y 333.732,Z 188.412,A -85,B 0,C 180,E1 -14426.247,E2 -14426.247} C_VEL
LIN {X 0,Y 333.688,Z 188.419,A -85,B 0,C 180,E1 -14428.975,E2 -14428.975} C_VEL
LIN {X 0,Y 333.642,Z 188.425,A -85,B 0,C 180,E1 -14432.588,E2 -14432.588} C_VEL
LIN {X 0,Y 333.684,Z 188.422,A -85,B 0,C 180,E1 -14434.775,E2 -14434.775} C_VEL
LIN {X 0,Y 333.815,Z 189.49,A -85,B 0,C 180,E1 -14436.868,E2 -14436.868} C_VEL
LIN {X 0,Y 334.279,Z 192.438,A -85,B 0,C 180,E1 -14440.811,E2 -14440.811} C_VEL
LIN {X 0,Y 334.672,Z 195.435,A -85,B 0,C 180,E1 -14444.441,E2 -14444.441} C_VEL
LIN {X 0,Y 334.899,Z 198.506,A -85,B 0,C 180,E1 -14447.815,E2 -14447.815} C_VEL
LIN {X 0,Y 334.835,Z 200.063,A -85,B 0,C 180,E1 -14449.408,E2 -14449.408} C_VEL
LIN {X 0,Y 334.351,Z 203.799,A -85,B 0,C 180,E1 -14453.012,E2 -14453.012} C_VEL
LIN {X 0,Y 333.752,Z 207.975,A -85,B 0,C 180,E1 -14456.805,E2 -14456.805} C_VEL
LIN {X 0,Y 333.214,Z 212.827,A -85,B 0,C 180,E1 -14460.981,E2 -14460.981} C_VEL
LIN {X 0,Y 332.864,Z 216.081,A -85,B 0,C 180,E1 -14463.68,E2 -14463.68} C_VEL
LIN {X 0,Y 332.614,Z 219.378,A -85,B 0,C 180,E1 -14466.331,E2 -14466.331} C_VEL
LIN {X 0,Y 332.47,Z 221.717,A -85,B 0,C 180,E1 -14468.159,E2 -14468.159} C_VEL
LIN {X 0,Y 334.828,Z 231.873,A -85,B 0,C 180,E1 -14468.709,E2 -14468.709} C_VEL
LIN {X 0,Y 336.602,Z 241.059,A -85,B 0,C 180,E1 -14469.313,E2 -14469.313} C_VEL
LIN {X 0,Y 337.863,Z 249.103,A -85,B 0,C 180,E1 -14469.927,E2 -14469.927} C_VEL
LIN {X 0,Y 338.994,Z 258.679,A -85,B 0,C 180,E1 -14470.785,E2 -14470.785} C_VEL
LIN {X 0,Y 339.128,Z 263.596,A -85,B 0,C 180,E1 -14471.264,E2 -14471.264} C_VEL
LIN {X 0,Y 337.651,Z 275.787,A -85,B 0,C 180,E1 -14472.59,E2 -14472.59} C_VEL
LIN {X 0,Y 336.474,Z 285.301,A -85,B 0,C 180,E1 -14473.909,E2 -14473.909} C_VEL
LIN {X 0,Y 335.569,Z 292.679,A -85,B 0,C 180,E1 -14475.134,E2 -14475.134} C_VEL
LIN {X 0,Y 334.776,Z 298.884,A -85,B 0,C 180,E1 -14476.339,E2 -14476.339} C_VEL
LIN {X 0,Y 333.85,Z 305.423,A -85,B 0,C 180,E1 -14477.848,E2 -14477.848} C_VEL
LIN {X 0,Y 333.352,Z 309.929,A -85,B 0,C 180,E1 -14479.062,E2 -14479.062} C_VEL
LIN {X 0,Y 332.678,Z 315.423,A -85,B 0,C 180,E1 -14480.884,E2 -14480.884} C_VEL
LIN {X 0,Y 332.281,Z 319.751,A -85,B 0,C 180,E1 -14482.709,E2 -14482.709} C_VEL
LIN {X 0,Y 332.074,Z 322.387,A -85,B 0,C 180,E1 -14484.106,E2 -14484.106} C_VEL
LIN {X 0,Y 332.006,Z 325.311,A -85,B 0,C 180,E1 -14486.359,E2 -14486.359} C_VEL
LIN {X 0,Y 331.917,Z 326.369,A -85,B 0,C 180,E1 -14487.573,E2 -14487.573} C_VEL
LIN {X 0,Y 331.905,Z 326.958,A -85,B 0,C 180,E1 -14488.787,E2 -14488.787} C_VEL
LIN {X 0,Y 331.905,Z 326.958,A -85,B 0,C 180,E1 -14491.213,E2 -14491.213} C_VEL
LIN {X 0,Y 331.917,Z 326.369,A -85,B 0,C 180,E1 -14492.427,E2 -14492.427} C_VEL
LIN {X 0,Y 332.021,Z 323.921,A -85,B 0,C 180,E1 -14494.857,E2 -14494.857} C_VEL
LIN {X 0,Y 332.185,Z 320.969,A -85,B 0,C 180,E1 -14496.682,E2 -14496.682} C_VEL
LIN {X 0,Y 332.513,Z 316.977,A -85,B 0,C 180,E1 -14498.508,E2 -14498.508} C_VEL
LIN {X 0,Y 333.086,Z 311.845,A -85,B 0,C 180,E1 -14500.332,E2 -14500.332} C_VEL
LIN {X 0,Y 333.695,Z 306.579,A -85,B 0,C 180,E1 -14501.85,E2 -14501.85} C_VEL
LIN {X 0,Y 334.568,Z 300.26,A -85,B 0,C 180,E1 -14503.36,E2 -14503.36} C_VEL
LIN {X 0,Y 335.349,Z 294.306,A -85,B 0,C 180,E1 -14504.565,E2 -14504.565} C_VEL
LIN {X 0,Y 336.408,Z 286.314,A -85,B 0,C 180,E1 -14505.931,E2 -14505.931} C_VEL
LIN {X 0,Y 337.331,Z 278.056,A -85,B 0,C 180,E1 -14507.114,E2 -14507.114} C_VEL
LIN {X 0,Y 338.428,Z 269.328,A -85,B 0,C 180,E1 -14508.149,E2 -14508.149} C_VEL
LIN {X 0,Y 339.222,Z 261.962,A -85,B 0,C 180,E1 -14508.888,E2 -14508.888} C_VEL
LIN {X 0,Y 338.254,Z 252.032,A -85,B 0,C 180,E1 -14509.82,E2 -14509.82} C_VEL
LIN {X 0,Y 336.968,Z 242.924,A -85,B 0,C 180,E1 -14510.549,E2 -14510.549} C_VEL
LIN {X 0,Y 334.953,Z 232.4,A -85,B 0,C 180,E1 -14511.259,E2 -14511.259} C_VEL
LIN {X 0,Y 332.467,Z 221.56,A -85,B 0,C 180,E1 -14511.885,E2 -14511.885} C_VEL
LIN {X 0,Y 332.741,Z 217.738,A -85,B 0,C 180,E1 -14514.988,E2 -14514.988} C_VEL
LIN {X 0,Y 333.062,Z 214.453,A -85,B 0,C 180,E1 -14517.66,E2 -14517.66} C_VEL
LIN {X 0,Y 333.547,Z 209.575,A -85,B 0,C 180,E1 -14521.786,E2 -14521.786} C_VEL
LIN {X 0,Y 334.026,Z 206.104,A -85,B 0,C 180,E1 -14524.857,E2 -14524.857} C_VEL
LIN {X 0,Y 334.403,Z 203.193,A -85,B 0,C 180,E1 -14527.551,E2 -14527.551} C_VEL
LIN {X 0,Y 334.858,Z 199.724,A -85,B 0,C 180,E1 -14530.924,E2 -14530.924} C_VEL
LIN {X 0,Y 334.831,Z 196.96,A -85,B 0,C 180,E1 -14533.84,E2 -14533.84} C_VEL
LIN {X 0,Y 334.447,Z 193.924,A -85,B 0,C 180,E1 -14537.347,E2 -14537.347} C_VEL
LIN {X 0,Y 334.054,Z 191.124,A -85,B 0,C 180,E1 -14540.864,E2 -14540.864} C_VEL
LIN {X 0,Y 333.755,Z 188.973,A -85,B 0,C 180,E1 -14543.87,E2 -14543.87} C_VEL
LIN {X 0,Y 333.672,Z 188.423,A -85,B 0,C 180,E1 -14545.34,E2 -14545.34} C_VEL
LIN {X 0,Y 333.688,Z 188.417,A -85,B 0,C 180,E1 -14549.636,E2 -14549.636} C_VEL
LIN {X 0,Y 333.737,Z 188.416,A -85,B 0,C 180,E1 -14552.4,E2 -14552.4} C_VEL
LIN {X 0,Y 333.724,Z 188.414,A -85,B 0,C 180,E1 -14555.09,E2 -14555.09} C_VEL
LIN {X 0,Y 333.677,Z 188.419,A -85,B 0,C 180,E1 -14559.018,E2 -14559.018} C_VEL
LIN {X 0,Y 333.79,Z 188.405,A -85,B 0,C 180,E1 -14561.589,E2 -14561.589} C_VEL
LIN {X 0,Y 333.805,Z 188.403,A -85,B 0,C 180,E1 -14565.576,E2 -14565.576} C_VEL
LIN {X 0,Y 333.83,Z 188.399,A -85,B 0,C 180,E1 -14569.077,E2 -14569.077} C_VEL
LIN {X 0,Y 334.001,Z 188.378,A -85,B 0,C 180,E1 -14572.746,E2 -14572.746} C_VEL
LIN {X 0,Y 333.802,Z 188.403,A -85,B 0,C 180,E1 -14575.168,E2 -14575.168} C_VEL
LIN {X 0,Y 334.099,Z 188.369,A -85,B 0,C 180,E1 -14577.588,E2 -14577.588} C_VEL
LIN {X 0,Y 334.242,Z 188.348,A -85,B 0,C 180,E1 -14579.999,E2 -14579.999} C_VEL
LIN {X 0,Y 334.1,Z 188.361,A -85,B 0,C 180,E1 -14582.411,E2 -14582.411} C_VEL
LIN {X 0,Y 333.987,Z 188.379,A -85,B 0,C 180,E1 -14586.654,E2 -14586.654} C_VEL
LIN {X 0,Y 333.845,Z 188.399,A -85,B 0,C 180,E1 -14589.695,E2 -14589.695} C_VEL
LIN {X 0,Y 333.791,Z 188.408,A -85,B 0,C 180,E1 -14593.391,E2 -14593.391} C_VEL
LIN {X 0,Y 333.741,Z 188.415,A -85,B 0,C 180,E1 -14597.146,E2 -14597.146} C_VEL
LIN {X 0,Y 333.733,Z 188.411,A -85,B 0,C 180,E1 -14599.69,E2 -14599.69} C_VEL
LIN {X 0,Y 333.687,Z 188.417,A -85,B 0,C 180,E1 -14602.278,E2 -14602.278} C_VEL
LIN {X 0,Y 333.73,Z 188.411,A -85,B 0,C 180,E1 -14606.246,E2 -14606.246} C_VEL
LIN {X 0,Y 333.706,Z 188.419,A -85,B 0,C 180,E1 -14608.972,E2 -14608.972} C_VEL
LIN {X 0,Y 333.638,Z 188.427,A -85,B 0,C 180,E1 -14612.587,E2 -14612.587} C_VEL
LIN {X 0,Y 333.671,Z 188.42,A -85,B 0,C 180,E1 -14616.139,E2 -14616.139} C_VEL
LIN {X 0,Y 333.667,Z 188.42,A -85,B 0,C 180,E1 -14619.189,E2 -14619.189} C_VEL
LIN {X 0,Y 333.655,Z 188.425,A -85,B 0,C 180,E1 -14622.505,E2 -14622.505} C_VEL
LIN {X 0,Y 333.591,Z 188.431,A -85,B 0,C 180,E1 -14625.955,E2 -14625.955} C_VEL
LIN {X 0,Y 333.642,Z 188.422,A -85,B 0,C 180,E1 -14629.315,E2 -14629.315} C_VEL
LIN {X 0,Y 333.66,Z 188.42,A -85,B 0,C 180,E1 -14633.168,E2 -14633.168} C_VEL
LIN {X 0,Y 333.637,Z 188.423,A -85,B 0,C 180,E1 -14636.792,E2 -14636.792} C_VEL
LIN {X 0,Y 333.7,Z 188.419,A -85,B 0,C 180,E1 -14639.71,E2 -14639.71} C_VEL
LIN {X 0,Y 333.74,Z 188.412,A -85,B 0,C 180,E1 -14642.401,E2 -14642.401} C_VEL
LIN {X 0,Y 333.722,Z 188.414,A -85,B 0,C 180,E1 -14645.091,E2 -14645.091} C_VEL
LIN {X 0,Y 333.705,Z 188.467,A -85,B 0,C 180,E1 -14648.779,E2 -14648.779} C_VEL
LIN {X 0,Y 334.6,Z 191.073,A -85,B 0,C 180,E1 -14648.988,E2 -14648.988} C_VEL
LIN {X 0,Y 336.957,Z 193.973,A -85,B 0,C 180,E1 -14649.431,E2 -14649.431} C_VEL
LIN {X 0,Y 339.211,Z 197.263,A -85,B 0,C 180,E1 -14649.878,E2 -14649.878} C_VEL
LIN {X 0,Y 340.84,Z 199.181,A -85,B 0,C 180,E1 -14650.199,E2 -14650.199} C_VEL
LIN {X 0,Y 343.892,Z 202.919,A -85,B 0,C 180,E1 -14650.82,E2 -14650.82} C_VEL
LIN {X 0,Y 348.4,Z 208.244,A -85,B 0,C 180,E1 -14651.783,E2 -14651.783} C_VEL
LIN {X 0,Y 350.501,Z 210.54,A -85,B 0,C 180,E1 -14652.254,E2 -14652.254} C_VEL
LIN {X 0,Y 354.225,Z 214.476,A -85,B 0,C 180,E1 -14653.111,E2 -14653.111} C_VEL
LIN {X 0,Y 359.545,Z 220.032,A -85,B 0,C 180,E1 -14654.434,E2 -14654.434} C_VEL
LIN {X 0,Y 362.602,Z 222.651,A -85,B 0,C 180,E1 -14655.236,E2 -14655.236} C_VEL
LIN {X 0,Y 366.37,Z 226.593,A -85,B 0,C 180,E1 -14656.351,E2 -14656.351} C_VEL
LIN {X 0,Y 370.103,Z 229.584,A -85,B 0,C 180,E1 -14657.519,E2 -14657.519} C_VEL
LIN {X 0,Y 373.301,Z 232.926,A -85,B 0,C 180,E1 -14658.694,E2 -14658.694} C_VEL
LIN {X 0,Y 376.874,Z 235.509,A -85,B 0,C 180,E1 -14660.07,E2 -14660.07} C_VEL
LIN {X 0,Y 378.655,Z 236.641,A -85,B 0,C 180,E1 -14660.836,E2 -14660.836} C_VEL
LIN {X 0,Y 381.453,Z 239.862,A -85,B 0,C 180,E1 -14662.375,E2 -14662.375} C_VEL
LIN {X 0,Y 383.848,Z 241.826,A -85,B 0,C 180,E1 -14663.891,E2 -14663.891} C_VEL
LIN {X 0,Y 386.042,Z 243.068,A -85,B 0,C 180,E1 -14665.615,E2 -14665.615} C_VEL
LIN {X 0,Y 387.269,Z 243.403,A -85,B 0,C 180,E1 -14666.879,E2 -14666.879} C_VEL
LIN {X 0,Y 387.975,Z 243.571,A -85,B 0,C 180,E1 -14667.924,E2 -14667.924} C_VEL
LIN {X 0,Y 388.423,Z 243.622,A -85,B 0,C 180,E1 -14668.963,E2 -14668.963} C_VEL
LIN {X 0,Y 388.571,Z 243.666,A -85,B 0,C 180,E1 -14670,E2 -14670} C_VEL
LIN {X 0,Y 388.419,Z 243.598,A -85,B 0,C 180,E1 -14671.037,E2 -14671.037} C_VEL
LIN {X 0,Y 387.275,Z 243.376,A -85,B 0,C 180,E1 -14673.121,E2 -14673.121} C_VEL
LIN {X 0,Y 385.349,Z 242.738,A -85,B 0,C 180,E1 -14674.979,E2 -14674.979} C_VEL
LIN {X 0,Y 382.745,Z 241.048,A -85,B 0,C 180,E1 -14676.835,E2 -14676.835} C_VEL
LIN {X 0,Y 379.98,Z 238.291,A -85,B 0,C 180,E1 -14678.453,E2 -14678.453} C_VEL
LIN {X 0,Y 378.17,Z 236.213,A -85,B 0,C 180,E1 -14679.366,E2 -14679.366} C_VEL
LIN {X 0,Y 375.135,Z 234.397,A -85,B 0,C 180,E1 -14680.599,E2 -14680.599} C_VEL
LIN {X 0,Y 371.825,Z 231.549,A -85,B 0,C 180,E1 -14681.856,E2 -14681.856} C_VEL
LIN {X 0,Y 369.184,Z 228.682,A -85,B 0,C 180,E1 -14682.793,E2 -14682.793} C_VEL
LIN {X 0,Y 365.487,Z 225.785,A -85,B 0,C 180,E1 -14683.914,E2 -14683.914} C_VEL
LIN {X 0,Y 361.345,Z 221.43,A -85,B 0,C 180,E1 -14685.109,E2 -14685.109} C_VEL
LIN {X 0,Y 357.492,Z 217.933,A -85,B 0,C 180,E1 -14686.106,E2 -14686.106} C_VEL
LIN {X 0,Y 354.404,Z 214.667,A -85,B 0,C 180,E1 -14686.846,E2 -14686.846} C_VEL
